LIN {X 0,Y 282.772,Z 519.685,A -85,B 0,C 180,E1 -19007.378,E2 -19007.378} C_VEL
LIN {X 0,Y 274.139,Z 501.017,A -85,B 0,C 180,E1 -19009.361,E2 -19009.361} C_VEL
LIN {X 0,Y 269.394,Z 492.351,A -85,B 0,C 180,E1 -19010.462,E2 -19010.462} C_VEL
LIN {X 0,Y 261.434,Z 479.486,A -85,B 0,C 180,E1 -19012.375,E2 -19012.375} C_VEL
LIN {X 0,Y 254.128,Z 468.54,A -85,B 0,C 180,E1 -19014.24,E2 -19014.24} C_VEL
LIN {X 0,Y 251.383,Z 464.398,A -85,B 0,C 180,E1 -19014.979,E2 -19014.979} C_VEL
LIN {X 0,Y 249.654,Z 462.021,A -85,B 0,C 180,E1 -19015.449,E2 -19015.449} C_VEL
LIN {X 0,Y 249.116,Z 460.076,A -85,B 0,C 180,E1 -19015.694,E2 -19015.694} C_VEL
LIN {X 0,Y 249.078,Z 460.074,A -85,B 0,C 180,E1 -19018.99,E2 -19018.99} C_VEL
LIN {X 0,Y 249.037,Z 460.072,A -85,B 0,C 180,E1 -19022.426,E2 -19022.426} C_VEL
LIN {X 0,Y 249.061,Z 460.079,A -85,B 0,C 180,E1 -19026.341,E2 -19026.341} C_VEL
LIN {X 0,Y 249.035,Z 460.089,A -85,B 0,C 180,E1 -19030.473,E2 -19030.473} C_VEL
LIN {X 0,Y 249.008,Z 460.09,A -85,B 0,C 180,E1 -19034.878,E2 -19034.878} C_VEL
LIN {X 0,Y 249.033,Z 460.078,A -85,B 0,C 180,E1 -19037.366,E2 -19037.366} C_VEL
LIN {X 0,Y 249.051,Z 460.087,A -85,B 0,C 180,E1 -19041.623,E2 -19041.623} C_VEL
LIN {X 0,Y 249.064,Z 460.077,A -85,B 0,C 180,E1 -19045.642,E2 -19045.642} C_VEL
LIN {X 0,Y 249.05,Z 460.069,A -85,B 0,C 180,E1 -19049.472,E2 -19049.472} C_VEL
LIN {X 0,Y 249.071,Z 460.084,A -85,B 0,C 180,E1 -19053.161,E2 -19053.161} C_VEL
LIN {X 0,Y 249.064,Z 460.062,A -85,B 0,C 180,E1 -19056.731,E2 -19056.731} C_VEL
LIN {X 0,Y 249.112,Z 460.078,A -85,B 0,C 180,E1 -19060.211,E2 -19060.211} C_VEL
LIN {X 0,Y 249.245,Z 460.04,A -85,B 0,C 180,E1 -19063.622,E2 -19063.622} C_VEL
LIN {X 0,Y 249.194,Z 460.062,A -85,B 0,C 180,E1 -19066.352,E2 -19066.352} C_VEL
LIN {X 0,Y 248.614,Z 460.143,A -85,B 0,C 180,E1 -19067.703,E2 -19067.703} C_VEL
LIN {X 0,Y 245.972,Z 460.48,A -85,B 0,C 180,E1 -19069.912,E2 -19069.912} C_VEL
LIN {X 0,Y 242.807,Z 460.868,A -85,B 0,C 180,E1 -19072.63,E2 -19072.63} C_VEL
LIN {X 0,Y 242.4,Z 460.912,A -85,B 0,C 180,E1 -19073.568,E2 -19073.568} C_VEL
LIN {X 0,Y 242.638,Z 460.869,A -85,B 0,C 180,E1 -19078.34,E2 -19078.34} C_VEL
LIN {X 0,Y 242.638,Z 460.881,A -85,B 0,C 180,E1 -19081.659,E2 -19081.659} C_VEL
LIN {X 0,Y 242.435,Z 460.897,A -85,B 0,C 180,E1 -19086.658,E2 -19086.658} C_VEL
LIN {X 0,Y 242.316,Z 460.916,A -85,B 0,C 180,E1 -19090.021,E2 -19090.021} C_VEL
LIN {X 0,Y 242.168,Z 460.944,A -85,B 0,C 180,E1 -19095.14,E2 -19095.14} C_VEL
LIN {X 0,Y 242.08,Z 460.932,A -85,B 0,C 180,E1 -19098.623,E2 -19098.623} C_VEL
LIN {X 0,Y 242.051,Z 460.957,A -85,B 0,C 180,E1 -19102.176,E2 -19102.176} C_VEL
LIN {X 0,Y 242.068,Z 460.953,A -85,B 0,C 180,E1 -19105.838,E2 -19105.838} C_VEL
LIN {X 0,Y 242.03,Z 460.962,A -85,B 0,C 180,E1 -19109.58,E2 -19109.58} C_VEL
LIN {X 0,Y 241.992,Z 460.962,A -85,B 0,C 180,E1 -19113.49,E2 -19113.49} C_VEL
LIN {X 0,Y 242.004,Z 460.963,A -85,B 0,C 180,E1 -19117.579,E2 -19117.579} C_VEL
LIN {X 0,Y 242.025,Z 461.128,A -85,B 0,C 180,E1 -19118.864,E2 -19118.864} C_VEL
LIN {X 0,Y 243.467,Z 465.75,A -85,B 0,C 180,E1 -19120.909,E2 -19120.909} C_VEL
LIN {X 0,Y 246.199,Z 470.197,A -85,B 0,C 180,E1 -19121.719,E2 -19121.719} C_VEL
LIN {X 0,Y 254.135,Z 483.567,A -85,B 0,C 180,E1 -19123.939,E2 -19123.939} C_VEL
LIN {X 0,Y 261.128,Z 496.498,A -85,B 0,C 180,E1 -19125.79,E2 -19125.79} C_VEL
LIN {X 0,Y 268.709,Z 512.001,A -85,B 0,C 180,E1 -19127.704,E2 -19127.704} C_VEL
LIN {X 0,Y 276.684,Z 530.632,A -85,B 0,C 180,E1 -19129.643,E2 -19129.643} C_VEL
LIN {X 0,Y 271.867,Z 629.009,A -85,B 0,C 180,E1 -19132.182,E2 -19132.182} C_VEL
LIN {X 0,Y 270.488,Z 644.739,A -85,B 0,C 180,E1 -19132.777,E2 -19132.777} C_VEL
LIN {X 0,Y 268.53,Z 659.205,A -85,B 0,C 180,E1 -19133.574,E2 -19133.574} C_VEL
LIN {X 0,Y 266.005,Z 673.975,A -85,B 0,C 180,E1 -19134.686,E2 -19134.686} C_VEL
LIN {X 0,Y 263.095,Z 688.32,A -85,B 0,C 180,E1 -19136.107,E2 -19136.107} C_VEL
LIN {X 0,Y 259.931,Z 701.339,A -85,B 0,C 180,E1 -19137.723,E2 -19137.723} C_VEL
LIN {X 0,Y 256.518,Z 714.469,A -85,B 0,C 180,E1 -19139.772,E2 -19139.772} C_VEL
LIN {X 0,Y 253.224,Z 725.427,A -85,B 0,C 180,E1 -19141.847,E2 -19141.847} C_VEL
LIN {X 0,Y 250.049,Z 736.273,A -85,B 0,C 180,E1 -19144.382,E2 -19144.382} C_VEL
LIN {X 0,Y 247.729,Z 744.182,A -85,B 0,C 180,E1 -19146.598,E2 -19146.598} C_VEL
LIN {X 0,Y 245.105,Z 752.602,A -85,B 0,C 180,E1 -19149.436,E2 -19149.436} C_VEL
LIN {X 0,Y 242.764,Z 760.654,A -85,B 0,C 180,E1 -19152.812,E2 -19152.812} C_VEL
LIN {X 0,Y 241.46,Z 766.039,A -85,B 0,C 180,E1 -19155.675,E2 -19155.675} C_VEL
LIN {X 0,Y 240.394,Z 771.037,A -85,B 0,C 180,E1 -19159.045,E2 -19159.045} C_VEL
LIN {X 0,Y 240.012,Z 773.943,A -85,B 0,C 180,E1 -19161.58,E2 -19161.58} C_VEL
LIN {X 0,Y 239.767,Z 776.64,A -85,B 0,C 180,E1 -19164.954,E2 -19164.954} C_VEL
LIN {X 0,Y 239.828,Z 778.136,A -85,B 0,C 180,E1 -19168.32,E2 -19168.32} C_VEL
LIN {X 0,Y 239.912,Z 778.446,A -85,B 0,C 180,E1 -19169.999,E2 -19169.999} C_VEL
LIN {X 0,Y 239.745,Z 778.19,A -85,B 0,C 180,E1 -19173.36,E2 -19173.36} C_VEL
LIN {X 0,Y 239.837,Z 776.785,A -85,B 0,C 180,E1 -19176.73,E2 -19176.73} C_VEL
LIN {X 0,Y 240.251,Z 774.162,A -85,B 0,C 180,E1 -19180.108,E2 -19180.108} C_VEL
LIN {X 0,Y 241.234,Z 770.329,A -85,B 0,C 180,E1 -19183.477,E2 -19183.477} C_VEL
LIN {X 0,Y 242.731,Z 765.203,A -85,B 0,C 180,E1 -19186.829,E2 -19186.829} C_VEL
LIN {X 0,Y 245.031,Z 758.665,A -85,B 0,C 180,E1 -19190.131,E2 -19190.131} C_VEL
LIN {X 0,Y 248.034,Z 750.541,A -85,B 0,C 180,E1 -19193.37,E2 -19193.37} C_VEL
LIN {X 0,Y 251.407,Z 741.915,A -85,B 0,C 180,E1 -19196.121,E2 -19196.121} C_VEL
LIN {X 0,Y 254.509,Z 733.203,A -85,B 0,C 180,E1 -19198.445,E2 -19198.445} C_VEL
LIN {X 0,Y 258.211,Z 722.949,A -85,B 0,C 180,E1 -19200.685,E2 -19200.685} C_VEL
LIN {X 0,Y 262.278,Z 710.731,A -85,B 0,C 180,E1 -19202.861,E2 -19202.861} C_VEL
LIN {X 0,Y 266.371,Z 697.186,A -85,B 0,C 180,E1 -19204.788,E2 -19204.788} C_VEL
LIN {X 0,Y 269.906,Z 683.486,A -85,B 0,C 180,E1 -19206.352,E2 -19206.352} C_VEL
LIN {X 0,Y 273.177,Z 668.696,A -85,B 0,C 180,E1 -19207.661,E2 -19207.661} C_VEL
LIN {X 0,Y 275.927,Z 654.171,A -85,B 0,C 180,E1 -19208.609,E2 -19208.609} C_VEL
LIN {X 0,Y 277.96,Z 639.385,A -85,B 0,C 180,E1 -19209.321,E2 -19209.321} C_VEL
LIN {X 0,Y 279.307,Z 622.797,A -85,B 0,C 180,E1 -19209.854,E2 -19209.854} C_VEL
LIN {X 0,Y 284.003,Z 540.814,A -85,B 0,C 180,E1 -19211.923,E2 -19211.923} C_VEL
LIN {X 0,Y 284.239,Z 534.234,A -85,B 0,C 180,E1 -19212.118,E2 -19212.118} C_VEL
LIN {X 0,Y 278.658,Z 520.932,A -85,B 0,C 180,E1 -19213.847,E2 -19213.847} C_VEL
LIN {X 0,Y 272.663,Z 508.788,A -85,B 0,C 180,E1 -19215.785,E2 -19215.785} C_VEL
LIN {X 0,Y 266.889,Z 498.341,A -85,B 0,C 180,E1 -19217.779,E2 -19217.779} C_VEL
LIN {X 0,Y 261.979,Z 490.421,A -85,B 0,C 180,E1 -19219.607,E2 -19219.607} C_VEL
LIN {X 0,Y 259.385,Z 486.385,A -85,B 0,C 180,E1 -19220.641,E2 -19220.641} C_VEL
LIN {X 0,Y 256.055,Z 481.339,A -85,B 0,C 180,E1 -19222.035,E2 -19222.035} C_VEL
LIN {X 0,Y 251.669,Z 475.022,A -85,B 0,C 180,E1 -19224.04,E2 -19224.04} C_VEL
LIN {X 0,Y 248.15,Z 470.216,A -85,B 0,C 180,E1 -19225.806,E2 -19225.806} C_VEL
LIN {X 0,Y 244.223,Z 465.374,A -85,B 0,C 180,E1 -19227.948,E2 -19227.948} C_VEL
LIN {X 0,Y 242.555,Z 462.973,A -85,B 0,C 180,E1 -19229.05,E2 -19229.05} C_VEL
LIN {X 0,Y 242.027,Z 460.958,A -85,B 0,C 180,E1 -19230.752,E2 -19230.752} C_VEL
LIN {X 0,Y 242.062,Z 460.956,A -85,B 0,C 180,E1 -19234.183,E2 -19234.183} C_VEL
LIN {X 0,Y 242.047,Z 460.958,A -85,B 0,C 180,E1 -19238.297,E2 -19238.297} C_VEL
LIN {X 0,Y 242.157,Z 460.935,A -85,B 0,C 180,E1 -19243.278,E2 -19243.278} C_VEL
LIN {X 0,Y 242.181,Z 460.942,A -85,B 0,C 180,E1 -19248.28,E2 -19248.28} C_VEL
LIN {X 0,Y 242.422,Z 460.909,A -85,B 0,C 180,E1 -19251.666,E2 -19251.666} C_VEL
LIN {X 0,Y 242.256,Z 460.926,A -85,B 0,C 180,E1 -19255.008,E2 -19255.008} C_VEL
LIN {X 0,Y 242.631,Z 460.878,A -85,B 0,C 180,E1 -19258.341,E2 -19258.341} C_VEL
LIN {X 0,Y 242.631,Z 460.877,A -85,B 0,C 180,E1 -19261.66,E2 -19261.66} C_VEL
LIN {X 0,Y 242.425,Z 460.912,A -85,B 0,C 180,E1 -19266.706,E2 -19266.706} C_VEL
LIN {X 0,Y 242.406,Z 461.074,A -85,B 0,C 180,E1 -19269.237,E2 -19269.237} C_VEL
LIN {X 0,Y 243.246,Z 463.656,A -85,B 0,C 180,E1 -19269.881,E2 -19269.881} C_VEL
LIN {X 0,Y 245.242,Z 465.908,A -85,B 0,C 180,E1 -19271.049,E2 -19271.049} C_VEL
LIN {X 0,Y 246.841,Z 466.95,A -85,B 0,C 180,E1 -19271.861,E2 -19271.861} C_VEL
LIN {X 0,Y 248.548,Z 470.005,A -85,B 0,C 180,E1 -19272.815,E2 -19272.815} C_VEL
LIN {X 0,Y 251.376,Z 472.668,A -85,B 0,C 180,E1 -19274.161,E2 -19274.161} C_VEL
LIN {X 0,Y 253.704,Z 476.012,A -85,B 0,C 180,E1 -19275.273,E2 -19275.273} C_VEL
LIN {X 0,Y 255.328,Z 477.907,A -85,B 0,C 180,E1 -19275.978,E2 -19275.978} C_VEL
LIN {X 0,Y 258.103,Z 481.555,A -85,B 0,C 180,E1 -19277.142,E2 -19277.142} C_VEL
LIN {X 0,Y 262.643,Z 487.86,A -85,B 0,C 180,E1 -19278.933,E2 -19278.933} C_VEL
LIN {X 0,Y 267.991,Z 495.314,A -85,B 0,C 180,E1 -19280.849,E2 -19280.849} C_VEL
LIN {X 0,Y 273.848,Z 504.485,A -85,B 0,C 180,E1 -19282.791,E2 -19282.791} C_VEL
LIN {X 0,Y 280.321,Z 516.959,A -85,B 0,C 180,E1 -19284.831,E2 -19284.831} C_VEL
LIN {X 0,Y 284.68,Z 526.585,A -85,B 0,C 180,E1 -19286.148,E2 -19286.148} C_VEL
LIN {X 0,Y 279.259,Z 620.067,A -85,B 0,C 180,E1 -19288.545,E2 -19288.545} C_VEL
LIN {X 0,Y 277.451,Z 636.178,A -85,B 0,C 180,E1 -19289.197,E2 -19289.197} C_VEL
LIN {X 0,Y 275.126,Z 651.64,A -85,B 0,C 180,E1 -19290.15,E2 -19290.15} C_VEL
LIN {X 0,Y 272.338,Z 665.875,A -85,B 0,C 180,E1 -19291.316,E2 -19291.316} C_VEL
LIN {X 0,Y 268.818,Z 680.57,A -85,B 0,C 180,E1 -19292.875,E2 -19292.875} C_VEL
LIN {X 0,Y 264.966,Z 694.127,A -85,B 0,C 180,E1 -19294.692,E2 -19294.692} C_VEL
LIN {X 0,Y 261.065,Z 706.563,A -85,B 0,C 180,E1 -19296.788,E2 -19296.788} C_VEL
LIN {X 0,Y 257.532,Z 716.783,A -85,B 0,C 180,E1 -19298.879,E2 -19298.879} C_VEL
LIN {X 0,Y 253.615,Z 727.436,A -85,B 0,C 180,E1 -19301.567,E2 -19301.567} C_VEL
LIN {X 0,Y 250.381,Z 735.735,A -85,B 0,C 180,E1 -19304.125,E2 -19304.125} C_VEL
LIN {X 0,Y 247.359,Z 743.322,A -85,B 0,C 180,E1 -19307.01,E2 -19307.01} C_VEL
LIN {X 0,Y 244.99,Z 749.256,A -85,B 0,C 180,E1 -19309.802,E2 -19309.802} C_VEL
LIN {X 0,Y 243.157,Z 754.125,A -85,B 0,C 180,E1 -19312.631,E2 -19312.631} C_VEL
LIN {X 0,Y 241.771,Z 757.966,A -85,B 0,C 180,E1 -19315.471,E2 -19315.471} C_VEL
LIN {X 0,Y 240.791,Z 760.856,A -85,B 0,C 180,E1 -19318.309,E2 -19318.309} C_VEL
LIN {X 0,Y 239.89,Z 763.38,A -85,B 0,C 180,E1 -19322.048,E2 -19322.048} C_VEL
LIN {X 0,Y 239.488,Z 764.479,A -85,B 0,C 180,E1 -19325.744,E2 -19325.744} C_VEL
LIN {X 0,Y 239.448,Z 764.232,A -85,B 0,C 180,E1 -19329.379,E2 -19329.379} C_VEL
LIN {X 0,Y 239.694,Z 762.699,A -85,B 0,C 180,E1 -19332.951,E2 -19332.951} C_VEL
LIN {X 0,Y 240.343,Z 759.891,A -85,B 0,C 180,E1 -19336.472,E2 -19336.472} C_VEL
LIN {X 0,Y 241.291,Z 755.788,A -85,B 0,C 180,E1 -19339.936,E2 -19339.936} C_VEL
LIN {X 0,Y 242.794,Z 750.301,A -85,B 0,C 180,E1 -19343.352,E2 -19343.352} C_VEL
LIN {X 0,Y 244.872,Z 743.309,A -85,B 0,C 180,E1 -19346.71,E2 -19346.71} C_VEL
LIN {X 0,Y 247.209,Z 735.768,A -85,B 0,C 180,E1 -19349.594,E2 -19349.594} C_VEL
LIN {X 0,Y 250.045,Z 726.708,A -85,B 0,C 180,E1 -19352.417,E2 -19352.417} C_VEL
LIN {X 0,Y 252.897,Z 717.459,A -85,B 0,C 180,E1 -19354.783,E2 -19354.783} C_VEL
LIN {X 0,Y 256.069,Z 706.558,A -85,B 0,C 180,E1 -19357.095,E2 -19357.095} C_VEL
LIN {X 0,Y 259.336,Z 694.632,A -85,B 0,C 180,E1 -19359.162,E2 -19359.162} C_VEL
LIN {X 0,Y 262.573,Z 681.588,A -85,B 0,C 180,E1 -19360.995,E2 -19360.995} C_VEL
LIN {X 0,Y 265.303,Z 668.808,A -85,B 0,C 180,E1 -19362.449,E2 -19362.449} C_VEL
LIN {X 0,Y 267.697,Z 655.458,A -85,B 0,C 180,E1 -19363.668,E2 -19363.668} C_VEL
LIN {X 0,Y 269.882,Z 640.363,A -85,B 0,C 180,E1 -19364.718,E2 -19364.718} C_VEL
LIN {X 0,Y 271.473,Z 626.008,A -85,B 0,C 180,E1 -19365.437,E2 -19365.437} C_VEL
LIN {X 0,Y 272.537,Z 610.439,A -85,B 0,C 180,E1 -19365.951,E2 -19365.951} C_VEL
LIN {X 0,Y 276.972,Z 521.758,A -85,B 0,C 180,E1 -19368.204,E2 -19368.204} C_VEL
LIN {X 0,Y 268.071,Z 502.626,A -85,B 0,C 180,E1 -19370.328,E2 -19370.328} C_VEL
LIN {X 0,Y 260.016,Z 488.824,A -85,B 0,C 180,E1 -19372.298,E2 -19372.298} C_VEL
LIN {X 0,Y 250.255,Z 473.861,A -85,B 0,C 180,E1 -19374.84,E2 -19374.84} C_VEL
LIN {X 0,Y 246.987,Z 469.165,A -85,B 0,C 180,E1 -19375.744,E2 -19375.744} C_VEL
LIN {X 0,Y 244.718,Z 465.681,A -85,B 0,C 180,E1 -19376.405,E2 -19376.405} C_VEL
LIN {X 0,Y 242.781,Z 463.346,A -85,B 0,C 180,E1 -19376.953,E2 -19376.953} C_VEL
LIN {X 0,Y 242.02,Z 460.953,A -85,B 0,C 180,E1 -19377.294,E2 -19377.294} C_VEL
LIN {X 0,Y 241.977,Z 460.958,A -85,B 0,C 180,E1 -19381.52,E2 -19381.52} C_VEL
LIN {X 0,Y 242.009,Z 460.965,A -85,B 0,C 180,E1 -19385.597,E2 -19385.597} C_VEL
LIN {X 0,Y 241.979,Z 460.959,A -85,B 0,C 180,E1 -19389.715,E2 -19389.715} C_VEL
LIN {X 0,Y 241.937,Z 460.963,A -85,B 0,C 180,E1 -19394.201,E2 -19394.201} C_VEL
LIN {X 0,Y 241.957,Z 460.954,A -85,B 0,C 180,E1 -19398.081,E2 -19398.081} C_VEL
LIN {X 0,Y 242.014,Z 460.958,A -85,B 0,C 180,E1 -19402.422,E2 -19402.422} C_VEL
LIN {X 0,Y 241.994,Z 460.966,A -85,B 0,C 180,E1 -19406.509,E2 -19406.509} C_VEL
LIN {X 0,Y 242.016,Z 460.944,A -85,B 0,C 180,E1 -19410.597,E2 -19410.597} C_VEL
LIN {X 0,Y 242.071,Z 460.954,A -85,B 0,C 180,E1 -19414.183,E2 -19414.183} C_VEL
LIN {X 0,Y 242.029,Z 460.95,A -85,B 0,C 180,E1 -19418.313,E2 -19418.313} C_VEL
LIN {X 0,Y 242.166,Z 460.921,A -85,B 0,C 180,E1 -19423.278,E2 -19423.278} C_VEL
LIN {X 0,Y 242.189,Z 460.934,A -85,B 0,C 180,E1 -19428.279,E2 -19428.279} C_VEL
LIN {X 0,Y 242.43,Z 460.896,A -85,B 0,C 180,E1 -19431.665,E2 -19431.665} C_VEL
LIN {X 0,Y 242.4,Z 460.912,A -85,B 0,C 180,E1 -19433.568,E2 -19433.568} C_VEL
LIN {X 0,Y 241.633,Z 461.006,A -85,B 0,C 180,E1 -19434.956,E2 -19434.956} C_VEL
LIN {X 0,Y 238.895,Z 461.343,A -85,B 0,C 180,E1 -19437.229,E2 -19437.229} C_VEL
LIN {X 0,Y 235.898,Z 461.726,A -85,B 0,C 180,E1 -19440.028,E2 -19440.028} C_VEL
LIN {X 0,Y 235.597,Z 461.756,A -85,B 0,C 180,E1 -19440.993,E2 -19440.993} C_VEL
LIN {X 0,Y 235.406,Z 461.776,A -85,B 0,C 180,E1 -19446.858,E2 -19446.858} C_VEL
LIN {X 0,Y 235.24,Z 461.792,A -85,B 0,C 180,E1 -19450.326,E2 -19450.326} C_VEL
LIN {X 0,Y 235.115,Z 461.824,A -85,B 0,C 180,E1 -19455.606,E2 -19455.606} C_VEL
LIN {X 0,Y 235.021,Z 461.812,A -85,B 0,C 180,E1 -19459.204,E2 -19459.204} C_VEL
LIN {X 0,Y 234.982,Z 461.835,A -85,B 0,C 180,E1 -19462.88,E2 -19462.88} C_VEL
LIN {X 0,Y 234.971,Z 461.841,A -85,B 0,C 180,E1 -19466.657,E2 -19466.657} C_VEL
LIN {X 0,Y 234.933,Z 461.842,A -85,B 0,C 180,E1 -19470.567,E2 -19470.567} C_VEL
LIN {X 0,Y 234.962,Z 461.843,A -85,B 0,C 180,E1 -19474.632,E2 -19474.632} C_VEL
LIN {X 0,Y 234.993,Z 461.954,A -85,B 0,C 180,E1 -19477.475,E2 -19477.475} C_VEL
LIN {X 0,Y 236.086,Z 465.459,A -85,B 0,C 180,E1 -19479.1,E2 -19479.1} C_VEL
LIN {X 0,Y 238.996,Z 470.175,A -85,B 0,C 180,E1 -19480.035,E2 -19480.035} C_VEL
LIN {X 0,Y 244.121,Z 478.587,A -85,B 0,C 180,E1 -19481.601,E2 -19481.601} C_VEL
LIN {X 0,Y 251.332,Z 490.98,A -85,B 0,C 180,E1 -19483.658,E2 -19483.658} C_VEL
LIN {X 0,Y 257.649,Z 503.054,A -85,B 0,C 180,E1 -19485.379,E2 -19485.379} C_VEL
LIN {X 0,Y 264.473,Z 517.44,A -85,B 0,C 180,E1 -19487.163,E2 -19487.163} C_VEL
LIN {X 0,Y 270.998,Z 532.796,A -85,B 0,C 180,E1 -19488.807,E2 -19488.807} C_VEL
LIN {X 0,Y 265.95,Z 630.58,A -85,B 0,C 180,E1 -19491.368,E2 -19491.368} C_VEL
LIN {X 0,Y 264.511,Z 645.629,A -85,B 0,C 180,E1 -19491.968,E2 -19491.968} C_VEL
LIN {X 0,Y 262.408,Z 660.442,A -85,B 0,C 180,E1 -19492.822,E2 -19492.822} C_VEL
LIN {X 0,Y 259.934,Z 674.242,A -85,B 0,C 180,E1 -19493.896,E2 -19493.896} C_VEL
LIN {X 0,Y 257.031,Z 687.913,A -85,B 0,C 180,E1 -19495.269,E2 -19495.269} C_VEL
LIN {X 0,Y 253.55,Z 701.866,A -85,B 0,C 180,E1 -19497.045,E2 -19497.045} C_VEL
LIN {X 0,Y 250.338,Z 713.789,A -85,B 0,C 180,E1 -19498.944,E2 -19498.944} C_VEL
LIN {X 0,Y 246.913,Z 724.827,A -85,B 0,C 180,E1 -19501.06,E2 -19501.06} C_VEL
LIN {X 0,Y 243.716,Z 735.267,A -85,B 0,C 180,E1 -19503.522,E2 -19503.522} C_VEL
LIN {X 0,Y 241.164,Z 743.679,A -85,B 0,C 180,E1 -19505.921,E2 -19505.921} C_VEL
LIN {X 0,Y 238.39,Z 752.151,A -85,B 0,C 180,E1 -19508.829,E2 -19508.829} C_VEL
LIN {X 0,Y 236.203,Z 759.359,A -85,B 0,C 180,E1 -19511.884,E2 -19511.884} C_VEL
LIN {X 0,Y 234.506,Z 765.677,A -85,B 0,C 180,E1 -19515.241,E2 -19515.241} C_VEL
LIN {X 0,Y 233.376,Z 770.716,A -85,B 0,C 180,E1 -19518.711,E2 -19518.711} C_VEL
LIN {X 0,Y 232.94,Z 773.639,A -85,B 0,C 180,E1 -19521.323,E2 -19521.323} C_VEL
LIN {X 0,Y 232.686,Z 776.373,A -85,B 0,C 180,E1 -19524.8,E2 -19524.8} C_VEL
LIN {X 0,Y 232.739,Z 777.903,A -85,B 0,C 180,E1 -19528.269,E2 -19528.269} C_VEL
LIN {X 0,Y 232.822,Z 778.23,A -85,B 0,C 180,E1 -19529.999,E2 -19529.999} C_VEL
LIN {X 0,Y 232.653,Z 778.005,A -85,B 0,C 180,E1 -19533.463,E2 -19533.463} C_VEL
LIN {X 0,Y 232.765,Z 776.622,A -85,B 0,C 180,E1 -19536.936,E2 -19536.936} C_VEL
LIN {X 0,Y 233.198,Z 774.024,A -85,B 0,C 180,E1 -19540.417,E2 -19540.417} C_VEL
LIN {X 0,Y 234.262,Z 770.229,A -85,B 0,C 180,E1 -19543.886,E2 -19543.886} C_VEL
LIN {X 0,Y 235.864,Z 765.15,A -85,B 0,C 180,E1 -19547.334,E2 -19547.334} C_VEL
LIN {X 0,Y 238.306,Z 758.66,A -85,B 0,C 180,E1 -19550.725,E2 -19550.725} C_VEL
LIN {X 0,Y 241.497,Z 750.583,A -85,B 0,C 180,E1 -19554.042,E2 -19554.042} C_VEL
LIN {X 0,Y 244.976,Z 742.009,A -85,B 0,C 180,E1 -19556.861,E2 -19556.861} C_VEL
LIN {X 0,Y 248.88,Z 731.737,A -85,B 0,C 180,E1 -19559.614,E2 -19559.614} C_VEL
LIN {X 0,Y 252.791,Z 721.28,A -85,B 0,C 180,E1 -19561.885,E2 -19561.885} C_VEL
LIN {X 0,Y 256.718,Z 709.956,A -85,B 0,C 180,E1 -19563.902,E2 -19563.902} C_VEL
LIN {X 0,Y 260.597,Z 697.687,A -85,B 0,C 180,E1 -19565.675,E2 -19565.675} C_VEL
LIN {X 0,Y 264.24,Z 684.24,A -85,B 0,C 180,E1 -19567.247,E2 -19567.247} C_VEL
LIN {X 0,Y 267.634,Z 669.612,A -85,B 0,C 180,E1 -19568.583,E2 -19568.583} C_VEL
LIN {X 0,Y 270.451,Z 655.394,A -85,B 0,C 180,E1 -19569.542,E2 -19569.542} C_VEL
LIN {X 0,Y 272.679,Z 640.192,A -85,B 0,C 180,E1 -19570.296,E2 -19570.296} C_VEL
LIN {X 0,Y 274.085,Z 624.371,A -85,B 0,C 180,E1 -19570.832,E2 -19570.832} C_VEL
LIN {X 0,Y 278.869,Z 544.481,A -85,B 0,C 180,E1 -19572.877,E2 -19572.877} C_VEL
LIN {X 0,Y 279.189,Z 536.605,A -85,B 0,C 180,E1 -19573.113,E2 -19573.113} C_VEL
LIN {X 0,Y 274.25,Z 524.669,A -85,B 0,C 180,E1 -19574.724,E2 -19574.724} C_VEL
LIN {X 0,Y 267.81,Z 511.374,A -85,B 0,C 180,E1 -19576.94,E2 -19576.94} C_VEL
LIN {X 0,Y 262.063,Z 501.21,A -85,B 0,C 180,E1 -19579.053,E2 -19579.053} C_VEL
LIN {X 0,Y 257.009,Z 492.813,A -85,B 0,C 180,E1 -19581.095,E2 -19581.095} C_VEL
LIN {X 0,Y 252.965,Z 486.736,A -85,B 0,C 180,E1 -19582.854,E2 -19582.854} C_VEL
LIN {X 0,Y 249.079,Z 480.95,A -85,B 0,C 180,E1 -19584.732,E2 -19584.732} C_VEL
LIN {X 0,Y 244.987,Z 475.331,A -85,B 0,C 180,E1 -19586.888,E2 -19586.888} C_VEL
LIN {X 0,Y 239.896,Z 468.74,A -85,B 0,C 180,E1 -19590.009,E2 -19590.009} C_VEL
LIN {X 0,Y 238.059,Z 466.791,A -85,B 0,C 180,E1 -19591.253,E2 -19591.253} C_VEL
LIN {X 0,Y 236.004,Z 464.746,A -85,B 0,C 180,E1 -19592.752,E2 -19592.752} C_VEL
LIN {X 0,Y 235.076,Z 462.308,A -85,B 0,C 180,E1 -19593.75,E2 -19593.75} C_VEL
LIN {X 0,Y 235.017,Z 461.836,A -85,B 0,C 180,E1 -19594.499,E2 -19594.499} C_VEL
LIN {X 0,Y 235.005,Z 461.829,A -85,B 0,C 180,E1 -19598.97,E2 -19598.97} C_VEL
LIN {X 0,Y 235.091,Z 461.815,A -85,B 0,C 180,E1 -19603.059,E2 -19603.059} C_VEL
LIN {X 0,Y 235.113,Z 461.818,A -85,B 0,C 180,E1 -19607.922,E2 -19607.922} C_VEL
LIN {X 0,Y 235.371,Z 461.784,A -85,B 0,C 180,E1 -19611.414,E2 -19611.414} C_VEL
LIN {X 0,Y 235.399,Z 461.781,A -85,B 0,C 180,E1 -19613.142,E2 -19613.142} C_VEL
LIN {X 0,Y 235.591,Z 461.754,A -85,B 0,C 180,E1 -19618.291,E2 -19618.291} C_VEL
LIN {X 0,Y 235.591,Z 461.754,A -85,B 0,C 180,E1 -19621.71,E2 -19621.71} C_VEL
LIN {X 0,Y 235.231,Z 461.943,A -85,B 0,C 180,E1 -19624.874,E2 -19624.874} C_VEL
LIN {X 0,Y 235.951,Z 464.084,A -85,B 0,C 180,E1 -19625.609,E2 -19625.609} C_VEL
LIN {X 0,Y 238.09,Z 466.548,A -85,B 0,C 180,E1 -19627.207,E2 -19627.207} C_VEL
LIN {X 0,Y 240.259,Z 467.791,A -85,B 0,C 180,E1 -19628.581,E2 -19628.581} C_VEL
LIN {X 0,Y 241.66,Z 470.698,A -85,B 0,C 180,E1 -19629.578,E2 -19629.578} C_VEL
LIN {X 0,Y 244.287,Z 473.107,A -85,B 0,C 180,E1 -19631.093,E2 -19631.093} C_VEL
LIN {X 0,Y 247.164,Z 477.235,A -85,B 0,C 180,E1 -19632.679,E2 -19632.679} C_VEL
LIN {X 0,Y 249.087,Z 479.099,A -85,B 0,C 180,E1 -19633.617,E2 -19633.617} C_VEL
LIN {X 0,Y 251.81,Z 482.758,A -85,B 0,C 180,E1 -19634.937,E2 -19634.937} C_VEL
LIN {X 0,Y 256.792,Z 489.477,A -85,B 0,C 180,E1 -19637.117,E2 -19637.117} C_VEL
LIN {X 0,Y 262.812,Z 498.023,A -85,B 0,C 180,E1 -19639.478,E2 -19639.478} C_VEL
LIN {X 0,Y 268.738,Z 507.04,A -85,B 0,C 180,E1 -19641.577,E2 -19641.577} C_VEL
LIN {X 0,Y 274.345,Z 517.578,A -85,B 0,C 180,E1 -19643.465,E2 -19643.465} C_VEL
LIN {X 0,Y 279.611,Z 528.887,A -85,B 0,C 180,E1 -19645.139,E2 -19645.139} C_VEL
LIN {X 0,Y 274.128,Z 620.295,A -85,B 0,C 180,E1 -19647.529,E2 -19647.529} C_VEL
LIN {X 0,Y 272.323,Z 636.028,A -85,B 0,C 180,E1 -19648.172,E2 -19648.172} C_VEL
LIN {X 0,Y 269.96,Z 651.279,A -85,B 0,C 180,E1 -19649.107,E2 -19649.107} C_VEL
LIN {X 0,Y 266.818,Z 666.703,A -85,B 0,C 180,E1 -19650.389,E2 -19650.389} C_VEL
LIN {X 0,Y 263.465,Z 680.303,A -85,B 0,C 180,E1 -19651.848,E2 -19651.848} C_VEL
LIN {X 0,Y 259.55,Z 693.614,A -85,B 0,C 180,E1 -19653.632,E2 -19653.632} C_VEL
LIN {X 0,Y 255.93,Z 704.914,A -85,B 0,C 180,E1 -19655.52,E2 -19655.52} C_VEL
LIN {X 0,Y 251.674,Z 716.605,A -85,B 0,C 180,E1 -19657.905,E2 -19657.905} C_VEL
LIN {X 0,Y 247.672,Z 727.043,A -85,B 0,C 180,E1 -19660.565,E2 -19660.565} C_VEL
LIN {X 0,Y 244.033,Z 735.932,A -85,B 0,C 180,E1 -19663.351,E2 -19663.351} C_VEL
LIN {X 0,Y 240.717,Z 743.827,A -85,B 0,C 180,E1 -19666.429,E2 -19666.429} C_VEL
LIN {X 0,Y 238.071,Z 750.096,A -85,B 0,C 180,E1 -19669.501,E2 -19669.501} C_VEL
LIN {X 0,Y 236.156,Z 754.814,A -85,B 0,C 180,E1 -19672.407,E2 -19672.407} C_VEL
LIN {X 0,Y 234.733,Z 758.576,A -85,B 0,C 180,E1 -19675.33,E2 -19675.33} C_VEL
LIN {X 0,Y 234.029,Z 760.54,A -85,B 0,C 180,E1 -19677.281,E2 -19677.281} C_VEL
LIN {X 0,Y 232.954,Z 763.307,A -85,B 0,C 180,E1 -19681.139,E2 -19681.139} C_VEL
LIN {X 0,Y 232.419,Z 764.636,A -85,B 0,C 180,E1 -19684.956,E2 -19684.956} C_VEL
LIN {X 0,Y 232.308,Z 764.599,A -85,B 0,C 180,E1 -19688.715,E2 -19688.715} C_VEL
LIN {X 0,Y 232.551,Z 763.252,A -85,B 0,C 180,E1 -19692.411,E2 -19692.411} C_VEL
LIN {X 0,Y 233.141,Z 760.632,A -85,B 0,C 180,E1 -19696.046,E2 -19696.046} C_VEL
LIN {X 0,Y 234.098,Z 756.726,A -85,B 0,C 180,E1 -19699.624,E2 -19699.624} C_VEL
LIN {X 0,Y 235.567,Z 751.469,A -85,B 0,C 180,E1 -19703.147,E2 -19703.147} C_VEL
LIN {X 0,Y 237.606,Z 744.741,A -85,B 0,C 180,E1 -19706.61,E2 -19706.61} C_VEL
LIN {X 0,Y 240.008,Z 737.369,A -85,B 0,C 180,E1 -19709.616,E2 -19709.616} C_VEL
LIN {X 0,Y 242.827,Z 728.716,A -85,B 0,C 180,E1 -19712.489,E2 -19712.489} C_VEL
LIN {X 0,Y 246.303,Z 718.004,A -85,B 0,C 180,E1 -19715.363,E2 -19715.363} C_VEL
LIN {X 0,Y 249.518,Z 707.369,A -85,B 0,C 180,E1 -19717.689,E2 -19717.689} C_VEL
LIN {X 0,Y 252.912,Z 695.548,A -85,B 0,C 180,E1 -19719.8,E2 -19719.8} C_VEL
LIN {X 0,Y 256.216,Z 682.661,A -85,B 0,C 180,E1 -19721.672,E2 -19721.672} C_VEL
LIN {X 0,Y 259.359,Z 668.478,A -85,B 0,C 180,E1 -19723.317,E2 -19723.317} C_VEL
LIN {X 0,Y 262.016,Z 653.89,A -85,B 0,C 180,E1 -19724.64,E2 -19724.64} C_VEL
LIN {X 0,Y 264.201,Z 638.736,A -85,B 0,C 180,E1 -19725.675,E2 -19725.675} C_VEL
LIN {X 0,Y 265.885,Z 623.254,A -85,B 0,C 180,E1 -19726.41,E2 -19726.41} C_VEL
LIN {X 0,Y 267.195,Z 602.123,A -85,B 0,C 180,E1 -19727.033,E2 -19727.033} C_VEL
LIN {X 0,Y 271.179,Z 523.87,A -85,B 0,C 180,E1 -19729.064,E2 -19729.064} C_VEL
LIN {X 0,Y 263.096,Z 506.355,A -85,B 0,C 180,E1 -19731.078,E2 -19731.078} C_VEL
LIN {X 0,Y 254.851,Z 492.324,A -85,B 0,C 180,E1 -19733.166,E2 -19733.166} C_VEL
LIN {X 0,Y 245.729,Z 478.276,A -85,B 0,C 180,E1 -19735.648,E2 -19735.648} C_VEL
LIN {X 0,Y 240.582,Z 470.787,A -85,B 0,C 180,E1 -19737.15,E2 -19737.15} C_VEL
LIN {X 0,Y 238.387,Z 467.61,A -85,B 0,C 180,E1 -19737.816,E2 -19737.816} C_VEL
LIN {X 0,Y 237.56,Z 466.5,A -85,B 0,C 180,E1 -19738.068,E2 -19738.068} C_VEL
LIN {X 0,Y 235.607,Z 464.055,A -85,B 0,C 180,E1 -19738.666,E2 -19738.666} C_VEL
LIN {X 0,Y 234.951,Z 461.833,A -85,B 0,C 180,E1 -19739.016,E2 -19739.016} C_VEL
LIN {X 0,Y 234.951,Z 461.827,A -85,B 0,C 180,E1 -19743.116,E2 -19743.116} C_VEL
LIN {X 0,Y 234.933,Z 461.831,A -85,B 0,C 180,E1 -19746.749,E2 -19746.749} C_VEL
LIN {X 0,Y 234.945,Z 461.826,A -85,B 0,C 180,E1 -19748.944,E2 -19748.944} C_VEL
LIN {X 0,Y 234.893,Z 461.837,A -85,B 0,C 180,E1 -19753.485,E2 -19753.485} C_VEL
LIN {X 0,Y 234.924,Z 461.845,A -85,B 0,C 180,E1 -19756.522,E2 -19756.522} C_VEL
LIN {X 0,Y 234.958,Z 461.843,A -85,B 0,C 180,E1 -19761.086,E2 -19761.086} C_VEL
LIN {X 0,Y 234.964,Z 461.831,A -85,B 0,C 180,E1 -19765.367,E2 -19765.367} C_VEL
LIN {X 0,Y 234.926,Z 461.828,A -85,B 0,C 180,E1 -19769.431,E2 -19769.431} C_VEL
LIN {X 0,Y 234.996,Z 461.837,A -85,B 0,C 180,E1 -19773.794,E2 -19773.794} C_VEL
LIN {X 0,Y 235.001,Z 461.833,A -85,B 0,C 180,E1 -19778.968,E2 -19778.968} C_VEL
LIN {X 0,Y 235.099,Z 461.802,A -85,B 0,C 180,E1 -19783.059,E2 -19783.059} C_VEL
LIN {X 0,Y 235.149,Z 461.813,A -85,B 0,C 180,E1 -19787.923,E2 -19787.923} C_VEL
LIN {X 0,Y 235.379,Z 461.771,A -85,B 0,C 180,E1 -19791.414,E2 -19791.414} C_VEL
LIN {X 0,Y 235.349,Z 461.789,A -85,B 0,C 180,E1 -19793.51,E2 -19793.51} C_VEL
LIN {X 0,Y 235.597,Z 461.745,A -85,B 0,C 180,E1 -19798.29,E2 -19798.29} C_VEL
LIN {X 0,Y 235.597,Z 461.756,A -85,B 0,C 180,E1 -19800.993,E2 -19800.993} C_VEL
LIN {X 0,Y 234.884,Z 461.842,A -85,B 0,C 180,E1 -19802.416,E2 -19802.416} C_VEL
LIN {X 0,Y 231.923,Z 462.206,A -85,B 0,C 180,E1 -19804.733,E2 -19804.733} C_VEL
LIN {X 0,Y 229.429,Z 462.517,A -85,B 0,C 180,E1 -19806.623,E2 -19806.623} C_VEL
LIN {X 0,Y 228.378,Z 462.663,A -85,B 0,C 180,E1 -19808.093,E2 -19808.093} C_VEL
LIN {X 0,Y 228.302,Z 462.668,A -85,B 0,C 180,E1 -19808.592,E2 -19808.592} C_VEL
LIN {X 0,Y 228.077,Z 462.672,A -85,B 0,C 180,E1 -19812.456,E2 -19812.456} C_VEL
LIN {X 0,Y 228.037,Z 462.689,A -85,B 0,C 180,E1 -19817.174,E2 -19817.174} C_VEL
LIN {X 0,Y 227.961,Z 462.712,A -85,B 0,C 180,E1 -19822.347,E2 -19822.347} C_VEL
LIN {X 0,Y 227.944,Z 462.715,A -85,B 0,C 180,E1 -19826.602,E2 -19826.602} C_VEL
LIN {X 0,Y 227.909,Z 462.718,A -85,B 0,C 180,E1 -19830.295,E2 -19830.295} C_VEL
LIN {X 0,Y 227.891,Z 462.719,A -85,B 0,C 180,E1 -19833.718,E2 -19833.718} C_VEL
LIN {X 0,Y 227.951,Z 462.886,A -85,B 0,C 180,E1 -19836.028,E2 -19836.028} C_VEL
LIN {X 0,Y 228.707,Z 465.217,A -85,B 0,C 180,E1 -19837.156,E2 -19837.156} C_VEL
LIN {X 0,Y 231.477,Z 469.647,A -85,B 0,C 180,E1 -19838.11,E2 -19838.11} C_VEL
LIN {X 0,Y 236.582,Z 477.781,A -85,B 0,C 180,E1 -19839.78,E2 -19839.78} C_VEL
LIN {X 0,Y 241.919,Z 486.668,A -85,B 0,C 180,E1 -19841.44,E2 -19841.44} C_VEL
LIN {X 0,Y 249.18,Z 499.721,A -85,B 0,C 180,E1 -19843.56,E2 -19843.56} C_VEL
LIN {X 0,Y 257.658,Z 516.902,A -85,B 0,C 180,E1 -19845.901,E2 -19845.901} C_VEL
LIN {X 0,Y 265.288,Z 534.93,A -85,B 0,C 180,E1 -19847.929,E2 -19847.929} C_VEL
LIN {X 0,Y 260.182,Z 630.385,A -85,B 0,C 180,E1 -19850.471,E2 -19850.471} C_VEL
LIN {X 0,Y 258.699,Z 645.428,A -85,B 0,C 180,E1 -19851.08,E2 -19851.08} C_VEL
LIN {X 0,Y 256.517,Z 660.233,A -85,B 0,C 180,E1 -19851.942,E2 -19851.942} C_VEL
LIN {X 0,Y 253.845,Z 674.742,A -85,B 0,C 180,E1 -19853.098,E2 -19853.098} C_VEL
LIN {X 0,Y 250.731,Z 688.757,A -85,B 0,C 180,E1 -19854.551,E2 -19854.551} C_VEL
LIN {X 0,Y 247.589,Z 701.022,A -85,B 0,C 180,E1 -19856.146,E2 -19856.146} C_VEL
LIN {X 0,Y 244.177,Z 713.055,A -85,B 0,C 180,E1 -19858.07,E2 -19858.07} C_VEL
LIN {X 0,Y 240.656,Z 724.191,A -85,B 0,C 180,E1 -19860.233,E2 -19860.233} C_VEL
LIN {X 0,Y 237.376,Z 734.36,A -85,B 0,C 180,E1 -19862.648,E2 -19862.648} C_VEL
LIN {X 0,Y 234.179,Z 744.498,A -85,B 0,C 180,E1 -19865.628,E2 -19865.628} C_VEL
LIN {X 0,Y 231.351,Z 752.825,A -85,B 0,C 180,E1 -19868.62,E2 -19868.62} C_VEL
LIN {X 0,Y 229.445,Z 758.77,A -85,B 0,C 180,E1 -19871.238,E2 -19871.238} C_VEL
LIN {X 0,Y 227.558,Z 765.315,A -85,B 0,C 180,E1 -19874.78,E2 -19874.78} C_VEL
LIN {X 0,Y 226.345,Z 770.393,A -85,B 0,C 180,E1 -19878.355,E2 -19878.355} C_VEL
LIN {X 0,Y 225.886,Z 773.336,A -85,B 0,C 180,E1 -19881.05,E2 -19881.05} C_VEL
LIN {X 0,Y 225.589,Z 776.106,A -85,B 0,C 180,E1 -19884.636,E2 -19884.636} C_VEL
LIN {X 0,Y 225.652,Z 777.671,A -85,B 0,C 180,E1 -19888.214,E2 -19888.214} C_VEL
LIN {X 0,Y 225.733,Z 778.013,A -85,B 0,C 180,E1 -19889.999,E2 -19889.999} C_VEL
LIN {X 0,Y 225.549,Z 777.821,A -85,B 0,C 180,E1 -19893.572,E2 -19893.572} C_VEL
LIN {X 0,Y 225.676,Z 776.457,A -85,B 0,C 180,E1 -19897.155,E2 -19897.155} C_VEL
LIN {X 0,Y 226.163,Z 773.896,A -85,B 0,C 180,E1 -19900.745,E2 -19900.745} C_VEL
LIN {X 0,Y 227.312,Z 770.141,A -85,B 0,C 180,E1 -19904.319,E2 -19904.319} C_VEL
LIN {X 0,Y 229.109,Z 764.851,A -85,B 0,C 180,E1 -19908.023,E2 -19908.023} C_VEL
LIN {X 0,Y 231.625,Z 758.656,A -85,B 0,C 180,E1 -19911.351,E2 -19911.351} C_VEL
LIN {X 0,Y 235.008,Z 750.634,A -85,B 0,C 180,E1 -19914.75,E2 -19914.75} C_VEL
LIN {X 0,Y 238.615,Z 742.136,A -85,B 0,C 180,E1 -19917.637,E2 -19917.637} C_VEL
LIN {X 0,Y 242.701,Z 731.947,A -85,B 0,C 180,E1 -19920.446,E2 -19920.446} C_VEL
LIN {X 0,Y 246.789,Z 721.57,A -85,B 0,C 180,E1 -19922.755,E2 -19922.755} C_VEL
LIN {X 0,Y 251.229,Z 709.18,A -85,B 0,C 180,E1 -19924.991,E2 -19924.991} C_VEL
LIN {X 0,Y 255.293,Z 696.804,A -85,B 0,C 180,E1 -19926.779,E2 -19926.779} C_VEL
LIN {X 0,Y 259.07,Z 683.343,A -85,B 0,C 180,E1 -19928.355,E2 -19928.355} C_VEL
LIN {X 0,Y 262.66,Z 668.407,A -85,B 0,C 180,E1 -19929.702,E2 -19929.702} C_VEL
LIN {X 0,Y 265.305,Z 655.339,A -85,B 0,C 180,E1 -19930.59,E2 -19930.59} C_VEL
LIN {X 0,Y 267.614,Z 640.245,A -85,B 0,C 180,E1 -19931.347,E2 -19931.347} C_VEL
LIN {X 0,Y 269.066,Z 624.672,A -85,B 0,C 180,E1 -19931.887,E2 -19931.887} C_VEL
LIN {X 0,Y 274.329,Z 540.453,A -85,B 0,C 180,E1 -19934.064,E2 -19934.064} C_VEL
LIN {X 0,Y 274.243,Z 538.891,A -85,B 0,C 180,E1 -19934.148,E2 -19934.148} C_VEL
LIN {X 0,Y 269.339,Z 527.123,A -85,B 0,C 180,E1 -19935.846,E2 -19935.846} C_VEL
LIN {X 0,Y 263.797,Z 515.619,A -85,B 0,C 180,E1 -19937.854,E2 -19937.854} C_VEL
LIN {X 0,Y 258.593,Z 506.174,A -85,B 0,C 180,E1 -19939.886,E2 -19939.886} C_VEL
LIN {X 0,Y 253.505,Z 497.661,A -85,B 0,C 180,E1 -19942.048,E2 -19942.048} C_VEL
LIN {X 0,Y 250.26,Z 492.545,A -85,B 0,C 180,E1 -19943.55,E2 -19943.55} C_VEL
LIN {X 0,Y 246.825,Z 487.243,A -85,B 0,C 180,E1 -19945.287,E2 -19945.287} C_VEL
LIN {X 0,Y 242.662,Z 481.485,A -85,B 0,C 180,E1 -19947.567,E2 -19947.567} C_VEL
LIN {X 0,Y 237.874,Z 475.023,A -85,B 0,C 180,E1 -19950.665,E2 -19950.665} C_VEL
LIN {X 0,Y 236.229,Z 473.351,A -85,B 0,C 180,E1 -19951.817,E2 -19951.817} C_VEL
LIN {X 0,Y 234.168,Z 471.004,A -85,B 0,C 180,E1 -19953.443,E2 -19953.443} C_VEL
LIN {X 0,Y 233.225,Z 468.702,A -85,B 0,C 180,E1 -19954.401,E2 -19954.401} C_VEL
LIN {X 0,Y 230.315,Z 467.212,A -85,B 0,C 180,E1 -19957.075,E2 -19957.075} C_VEL
LIN {X 0,Y 228.301,Z 464.25,A -85,B 0,C 180,E1 -19959.738,E2 -19959.738} C_VEL
LIN {X 0,Y 227.959,Z 462.707,A -85,B 0,C 180,E1 -19960.528,E2 -19960.528} C_VEL
LIN {X 0,Y 228.052,Z 462.694,A -85,B 0,C 180,E1 -19963.898,E2 -19963.898} C_VEL
LIN {X 0,Y 228.069,Z 462.692,A -85,B 0,C 180,E1 -19967.543,E2 -19967.543} C_VEL
LIN {X 0,Y 228.3,Z 462.663,A -85,B 0,C 180,E1 -19971.146,E2 -19971.146} C_VEL
LIN {X 0,Y 228.35,Z 462.661,A -85,B 0,C 180,E1 -19972.929,E2 -19972.929} C_VEL
LIN {X 0,Y 228.568,Z 462.656,A -85,B 0,C 180,E1 -19978.789,E2 -19978.789} C_VEL
LIN {X 0,Y 229.125,Z 464.582,A -85,B 0,C 180,E1 -19979.781,E2 -19979.781} C_VEL
LIN {X 0,Y 231.369,Z 467.581,A -85,B 0,C 180,E1 -19982.395,E2 -19982.395} C_VEL
LIN {X 0,Y 233.53,Z 468.883,A -85,B 0,C 180,E1 -19984.315,E2 -19984.315} C_VEL
LIN {X 0,Y 235.002,Z 471.74,A -85,B 0,C 180,E1 -19985.686,E2 -19985.686} C_VEL
LIN {X 0,Y 237.748,Z 474.097,A -85,B 0,C 180,E1 -19987.645,E2 -19987.645} C_VEL
LIN {X 0,Y 238.434,Z 474.741,A -85,B 0,C 180,E1 -19988.102,E2 -19988.102} C_VEL
LIN {X 0,Y 240.246,Z 477.803,A -85,B 0,C 180,E1 -19989.365,E2 -19989.365} C_VEL
LIN {X 0,Y 242.642,Z 480.19,A -85,B 0,C 180,E1 -19990.788,E2 -19990.788} C_VEL
LIN {X 0,Y 245.107,Z 483.695,A -85,B 0,C 180,E1 -19992.189,E2 -19992.189} C_VEL
LIN {X 0,Y 246.802,Z 485.456,A -85,B 0,C 180,E1 -19993.051,E2 -19993.051} C_VEL
LIN {X 0,Y 250.562,Z 490.646,A -85,B 0,C 180,E1 -19994.915,E2 -19994.915} C_VEL
LIN {X 0,Y 254.109,Z 495.492,A -85,B 0,C 180,E1 -19996.508,E2 -19996.508} C_VEL
LIN {X 0,Y 261.386,Z 506.051,A -85,B 0,C 180,E1 -19999.435,E2 -19999.435} C_VEL
LIN {X 0,Y 266.956,Z 515.278,A -85,B 0,C 180,E1 -20001.464,E2 -20001.464} C_VEL
LIN {X 0,Y 272.45,Z 526.474,A -85,B 0,C 180,E1 -20003.372,E2 -20003.372} C_VEL
LIN {X 0,Y 274.687,Z 531.463,A -85,B 0,C 180,E1 -20004.115,E2 -20004.115} C_VEL
LIN {X 0,Y 269.139,Z 620.258,A -85,B 0,C 180,E1 -20006.459,E2 -20006.459} C_VEL
LIN {X 0,Y 267.243,Z 636.44,A -85,B 0,C 180,E1 -20007.126,E2 -20007.126} C_VEL
LIN {X 0,Y 264.805,Z 651.517,A -85,B 0,C 180,E1 -20008.062,E2 -20008.062} C_VEL
LIN {X 0,Y 261.716,Z 666.222,A -85,B 0,C 180,E1 -20009.288,E2 -20009.288} C_VEL
LIN {X 0,Y 258.16,Z 680.099,A -85,B 0,C 180,E1 -20010.779,E2 -20010.779} C_VEL
LIN {X 0,Y 254.224,Z 693.096,A -85,B 0,C 180,E1 -20012.526,E2 -20012.526} C_VEL
LIN {X 0,Y 250.434,Z 704.466,A -85,B 0,C 180,E1 -20014.436,E2 -20014.436} C_VEL
LIN {X 0,Y 245.897,Z 716.435,A -85,B 0,C 180,E1 -20016.885,E2 -20016.885} C_VEL
LIN {X 0,Y 242.062,Z 726.041,A -85,B 0,C 180,E1 -20019.344,E2 -20019.344} C_VEL
LIN {X 0,Y 238.497,Z 734.356,A -85,B 0,C 180,E1 -20021.923,E2 -20021.923} C_VEL
LIN {X 0,Y 235.124,Z 741.913,A -85,B 0,C 180,E1 -20024.776,E2 -20024.776} C_VEL
LIN {X 0,Y 231.95,Z 749.126,A -85,B 0,C 180,E1 -20028.197,E2 -20028.197} C_VEL
LIN {X 0,Y 229.752,Z 754.119,A -85,B 0,C 180,E1 -20031.166,E2 -20031.166} C_VEL
LIN {X 0,Y 228.102,Z 758.021,A -85,B 0,C 180,E1 -20034.17,E2 -20034.17} C_VEL
LIN {X 0,Y 227.132,Z 760.592,A -85,B 0,C 180,E1 -20036.663,E2 -20036.663} C_VEL
LIN {X 0,Y 225.989,Z 763.369,A -85,B 0,C 180,E1 -20040.549,E2 -20040.549} C_VEL
LIN {X 0,Y 225.338,Z 764.846,A -85,B 0,C 180,E1 -20044.753,E2 -20044.753} C_VEL
LIN {X 0,Y 225.265,Z 764.618,A -85,B 0,C 180,E1 -20049.386,E2 -20049.386} C_VEL
LIN {X 0,Y 225.384,Z 763.743,A -85,B 0,C 180,E1 -20051.832,E2 -20051.832} C_VEL
LIN {X 0,Y 225.959,Z 761.339,A -85,B 0,C 180,E1 -20055.593,E2 -20055.593} C_VEL
LIN {X 0,Y 226.884,Z 757.655,A -85,B 0,C 180,E1 -20059.29,E2 -20059.29} C_VEL
LIN {X 0,Y 228.326,Z 752.63,A -85,B 0,C 180,E1 -20062.929,E2 -20062.929} C_VEL
LIN {X 0,Y 230.354,Z 746.15,A -85,B 0,C 180,E1 -20066.503,E2 -20066.503} C_VEL
LIN {X 0,Y 232.565,Z 739.775,A -85,B 0,C 180,E1 -20069.323,E2 -20069.323} C_VEL
LIN {X 0,Y 235.65,Z 730.687,A -85,B 0,C 180,E1 -20072.565,E2 -20072.565} C_VEL
LIN {X 0,Y 239.061,Z 720.498,A -85,B 0,C 180,E1 -20075.484,E2 -20075.484} C_VEL
LIN {X 0,Y 242.458,Z 710.038,A -85,B 0,C 180,E1 -20077.924,E2 -20077.924} C_VEL
LIN {X 0,Y 246.137,Z 697.606,A -85,B 0,C 180,E1 -20080.281,E2 -20080.281} C_VEL
LIN {X 0,Y 249.553,Z 685.091,A -85,B 0,C 180,E1 -20082.194,E2 -20082.194} C_VEL
LIN {X 0,Y 252.812,Z 671.405,A -85,B 0,C 180,E1 -20083.874,E2 -20083.874} C_VEL
LIN {X 0,Y 255.536,Z 657.526,A -85,B 0,C 180,E1 -20085.227,E2 -20085.227} C_VEL
LIN {X 0,Y 258.002,Z 642.051,A -85,B 0,C 180,E1 -20086.366,E2 -20086.366} C_VEL
LIN {X 0,Y 259.798,Z 627.006,A -85,B 0,C 180,E1 -20087.16,E2 -20087.16} C_VEL
LIN {X 0,Y 260.96,Z 611.265,A -85,B 0,C 180,E1 -20087.703,E2 -20087.703} C_VEL
LIN {X 0,Y 265.575,Z 526.542,A -85,B 0,C 180,E1 -20089.913,E2 -20089.913} C_VEL
LIN {X 0,Y 259.895,Z 513.709,A -85,B 0,C 180,E1 -20091.395,E2 -20091.395} C_VEL
LIN {X 0,Y 255.603,Z 505.585,A -85,B 0,C 180,E1 -20092.509,E2 -20092.509} C_VEL
LIN {X 0,Y 247.152,Z 491.641,A -85,B 0,C 180,E1 -20094.786,E2 -20094.786} C_VEL
LIN {X 0,Y 238.764,Z 478.936,A -85,B 0,C 180,E1 -20097.228,E2 -20097.228} C_VEL
LIN {X 0,Y 233.763,Z 471.904,A -85,B 0,C 180,E1 -20098.779,E2 -20098.779} C_VEL
LIN {X 0,Y 231.484,Z 468.626,A -85,B 0,C 180,E1 -20099.527,E2 -20099.527} C_VEL
LIN {X 0,Y 230.644,Z 467.459,A -85,B 0,C 180,E1 -20099.807,E2 -20099.807} C_VEL
LIN {X 0,Y 228.73,Z 465.249,A -85,B 0,C 180,E1 -20100.435,E2 -20100.435} C_VEL
LIN {X 0,Y 227.876,Z 462.722,A -85,B 0,C 180,E1 -20100.827,E2 -20100.827} C_VEL
LIN {X 0,Y 227.884,Z 462.711,A -85,B 0,C 180,E1 -20103.72,E2 -20103.72} C_VEL
LIN {X 0,Y 227.87,Z 462.704,A -85,B 0,C 180,E1 -20108.087,E2 -20108.087} C_VEL
LIN {X 0,Y 227.821,Z 462.719,A -85,B 0,C 180,E1 -20112.741,E2 -20112.741} C_VEL
LIN {X 0,Y 227.851,Z 462.716,A -85,B 0,C 180,E1 -20117.266,E2 -20117.266} C_VEL
LIN {X 0,Y 227.874,Z 462.722,A -85,B 0,C 180,E1 -20121.914,E2 -20121.914} C_VEL
LIN {X 0,Y 227.894,Z 462.722,A -85,B 0,C 180,E1 -20126.373,E2 -20126.373} C_VEL
LIN {X 0,Y 227.907,Z 462.7,A -85,B 0,C 180,E1 -20130.436,E2 -20130.436} C_VEL
LIN {X 0,Y 227.927,Z 462.715,A -85,B 0,C 180,E1 -20134.425,E2 -20134.425} C_VEL
LIN {X 0,Y 227.95,Z 462.701,A -85,B 0,C 180,E1 -20138.285,E2 -20138.285} C_VEL
LIN {X 0,Y 228.037,Z 462.682,A -85,B 0,C 180,E1 -20142.826,E2 -20142.826} C_VEL
LIN {X 0,Y 228.096,Z 462.694,A -85,B 0,C 180,E1 -20147.544,E2 -20147.544} C_VEL
LIN {X 0,Y 228.308,Z 462.649,A -85,B 0,C 180,E1 -20151.146,E2 -20151.146} C_VEL
LIN {X 0,Y 228.357,Z 462.662,A -85,B 0,C 180,E1 -20152.928,E2 -20152.928} C_VEL
LIN {X 0,Y 228.556,Z 462.621,A -85,B 0,C 180,E1 -20158.237,E2 -20158.237} C_VEL
LIN {X 0,Y 228.556,Z 462.634,A -85,B 0,C 180,E1 -20161.762,E2 -20161.762} C_VEL
LIN {X 0,Y 228.357,Z 462.657,A -85,B 0,C 180,E1 -20167.071,E2 -20167.071} C_VEL
LIN {X 0,Y 228.302,Z 462.668,A -85,B 0,C 180,E1 -20168.592,E2 -20168.592} C_VEL
LIN {X 0,Y 227.984,Z 462.715,A -85,B 0,C 180,E1 -20169.575,E2 -20169.575} C_VEL
LIN {X 0,Y 226.582,Z 462.892,A -85,B 0,C 180,E1 -20171.024,E2 -20171.024} C_VEL
LIN {X 0,Y 222.097,Z 463.438,A -85,B 0,C 180,E1 -20174.407,E2 -20174.407} C_VEL
LIN {X 0,Y 221.063,Z 463.572,A -85,B 0,C 180,E1 -20175.928,E2 -20175.928} C_VEL
LIN {X 0,Y 221.006,Z 463.571,A -85,B 0,C 180,E1 -20176.444,E2 -20176.444} C_VEL
LIN {X 0,Y 220.911,Z 463.583,A -85,B 0,C 180,E1 -20180.484,E2 -20180.484} C_VEL
LIN {X 0,Y 220.874,Z 463.598,A -85,B 0,C 180,E1 -20184.434,E2 -20184.434} C_VEL
LIN {X 0,Y 220.837,Z 463.597,A -85,B 0,C 180,E1 -20188.513,E2 -20188.513} C_VEL
LIN {X 0,Y 220.825,Z 463.601,A -85,B 0,C 180,E1 -20192.754,E2 -20192.754} C_VEL
LIN {X 0,Y 220.837,Z 463.64,A -85,B 0,C 180,E1 -20194.354,E2 -20194.354} C_VEL
LIN {X 0,Y 221.06,Z 464.728,A -85,B 0,C 180,E1 -20194.908,E2 -20194.908} C_VEL
LIN {X 0,Y 222.373,Z 467.158,A -85,B 0,C 180,E1 -20195.432,E2 -20195.432} C_VEL
LIN {X 0,Y 225.305,Z 471.087,A -85,B 0,C 180,E1 -20196.489,E2 -20196.489} C_VEL
LIN {X 0,Y 229.125,Z 477.165,A -85,B 0,C 180,E1 -20197.84,E2 -20197.84} C_VEL
LIN {X 0,Y 233.313,Z 483.952,A -85,B 0,C 180,E1 -20199.24,E2 -20199.24} C_VEL
LIN {X 0,Y 240.234,Z 495.769,A -85,B 0,C 180,E1 -20201.439,E2 -20201.439} C_VEL
LIN {X 0,Y 247.149,Z 508.987,A -85,B 0,C 180,E1 -20203.507,E2 -20203.507} C_VEL
LIN {X 0,Y 254.515,Z 524.703,A -85,B 0,C 180,E1 -20205.601,E2 -20205.601} C_VEL
LIN {X 0,Y 259.686,Z 537.134,A -85,B 0,C 180,E1 -20207.024,E2 -20207.024} C_VEL
LIN {X 0,Y 254.244,Z 632.938,A -85,B 0,C 180,E1 -20209.618,E2 -20209.618} C_VEL
LIN {X 0,Y 252.526,Z 648.685,A -85,B 0,C 180,E1 -20210.329,E2 -20210.329} C_VEL
LIN {X 0,Y 250.053,Z 663.786,A -85,B 0,C 180,E1 -20211.291,E2 -20211.291} C_VEL
LIN {X 0,Y 247.108,Z 678.4,A -85,B 0,C 180,E1 -20212.56,E2 -20212.56} C_VEL
LIN {X 0,Y 243.724,Z 692.555,A -85,B 0,C 180,E1 -20214.161,E2 -20214.161} C_VEL
LIN {X 0,Y 240.2,Z 705.314,A -85,B 0,C 180,E1 -20215.973,E2 -20215.973} C_VEL
LIN {X 0,Y 236.421,Z 717.664,A -85,B 0,C 180,E1 -20218.153,E2 -20218.153} C_VEL
LIN {X 0,Y 232.653,Z 728.926,A -85,B 0,C 180,E1 -20220.601,E2 -20220.601} C_VEL
LIN {X 0,Y 229.488,Z 738.422,A -85,B 0,C 180,E1 -20223.146,E2 -20223.146} C_VEL
LIN {X 0,Y 226.705,Z 746.482,A -85,B 0,C 180,E1 -20225.747,E2 -20225.747} C_VEL
LIN {X 0,Y 223.959,Z 754.429,A -85,B 0,C 180,E1 -20228.845,E2 -20228.845} C_VEL
LIN {X 0,Y 221.81,Z 760.833,A -85,B 0,C 180,E1 -20231.904,E2 -20231.904} C_VEL
LIN {X 0,Y 220.285,Z 766.383,A -85,B 0,C 180,E1 -20235.212,E2 -20235.212} C_VEL
LIN {X 0,Y 219.136,Z 771.143,A -85,B 0,C 180,E1 -20238.905,E2 -20238.905} C_VEL
LIN {X 0,Y 218.618,Z 774.584,A -85,B 0,C 180,E1 -20242.611,E2 -20242.611} C_VEL
LIN {X 0,Y 218.45,Z 776.781,A -85,B 0,C 180,E1 -20246.31,E2 -20246.31} C_VEL
LIN {X 0,Y 218.647,Z 777.796,A -85,B 0,C 180,E1 -20249.999,E2 -20249.999} C_VEL
LIN {X 0,Y 218.448,Z 777.64,A -85,B 0,C 180,E1 -20253.688,E2 -20253.688} C_VEL
LIN {X 0,Y 218.601,Z 776.294,A -85,B 0,C 180,E1 -20257.388,E2 -20257.388} C_VEL
LIN {X 0,Y 219.146,Z 773.769,A -85,B 0,C 180,E1 -20261.093,E2 -20261.093} C_VEL
LIN {X 0,Y 220.383,Z 770.053,A -85,B 0,C 180,E1 -20264.779,E2 -20264.779} C_VEL
LIN {X 0,Y 222.205,Z 765.06,A -85,B 0,C 180,E1 -20268.437,E2 -20268.437} C_VEL
LIN {X 0,Y 224.992,Z 758.674,A -85,B 0,C 180,E1 -20272.013,E2 -20272.013} C_VEL
LIN {X 0,Y 228.562,Z 750.713,A -85,B 0,C 180,E1 -20275.497,E2 -20275.497} C_VEL
LIN {X 0,Y 232.446,Z 741.889,A -85,B 0,C 180,E1 -20278.577,E2 -20278.577} C_VEL
LIN {X 0,Y 236.595,Z 732.156,A -85,B 0,C 180,E1 -20281.319,E2 -20281.319} C_VEL
LIN {X 0,Y 240.837,Z 721.869,A -85,B 0,C 180,E1 -20283.671,E2 -20283.671} C_VEL
LIN {X 0,Y 245.458,Z 709.615,A -85,B 0,C 180,E1 -20285.94,E2 -20285.94} C_VEL
LIN {X 0,Y 249.667,Z 697.384,A -85,B 0,C 180,E1 -20287.751,E2 -20287.751} C_VEL
LIN {X 0,Y 253.541,Z 684.243,A -85,B 0,C 180,E1 -20289.325,E2 -20289.325} C_VEL
LIN {X 0,Y 257.274,Z 669.458,A -85,B 0,C 180,E1 -20290.706,E2 -20290.706} C_VEL
LIN {X 0,Y 259.984,Z 656.628,A -85,B 0,C 180,E1 -20291.603,E2 -20291.603} C_VEL
LIN {X 0,Y 262.376,Z 642.13,A -85,B 0,C 180,E1 -20292.362,E2 -20292.362} C_VEL
LIN {X 0,Y 264.058,Z 626.387,A -85,B 0,C 180,E1 -20292.935,E2 -20292.935} C_VEL
LIN {X 0,Y 269.511,Z 542.713,A -85,B 0,C 180,E1 -20295.132,E2 -20295.132} C_VEL
LIN {X 0,Y 269.399,Z 541.268,A -85,B 0,C 180,E1 -20295.222,E2 -20295.222} C_VEL
LIN {X 0,Y 264.802,Z 530.259,A -85,B 0,C 180,E1 -20296.908,E2 -20296.908} C_VEL
LIN {X 0,Y 260.161,Z 520.429,A -85,B 0,C 180,E1 -20298.697,E2 -20298.697} C_VEL
LIN {X 0,Y 255.606,Z 511.867,A -85,B 0,C 180,E1 -20300.565,E2 -20300.565} C_VEL
LIN {X 0,Y 250.63,Z 503.288,A -85,B 0,C 180,E1 -20302.786,E2 -20302.786} C_VEL
LIN {X 0,Y 247.042,Z 497.512,A -85,B 0,C 180,E1 -20304.549,E2 -20304.549} C_VEL
LIN {X 0,Y 244.318,Z 493.199,A -85,B 0,C 180,E1 -20305.998,E2 -20305.998} C_VEL
LIN {X 0,Y 240.53,Z 487.727,A -85,B 0,C 180,E1 -20308.19,E2 -20308.19} C_VEL
LIN {X 0,Y 235.741,Z 481.09,A -85,B 0,C 180,E1 -20311.44,E2 -20311.44} C_VEL
LIN {X 0,Y 232.778,Z 477.965,A -85,B 0,C 180,E1 -20313.761,E2 -20313.761} C_VEL
LIN {X 0,Y 231.683,Z 475.642,A -85,B 0,C 180,E1 -20314.87,E2 -20314.87} C_VEL
LIN {X 0,Y 228.65,Z 473.681,A -85,B 0,C 180,E1 -20317.852,E2 -20317.852} C_VEL
LIN {X 0,Y 226.924,Z 470.62,A -85,B 0,C 180,E1 -20320.436,E2 -20320.436} C_VEL
LIN {X 0,Y 226.653,Z 469.689,A -85,B 0,C 180,E1 -20321,E2 -20321} C_VEL
LIN {X 0,Y 224.012,Z 468.467,A -85,B 0,C 180,E1 -20329.15,E2 -20329.15} C_VEL
LIN {X 0,Y 224.797,Z 468.873,A -85,B 0,C 180,E1 -20333.718,E2 -20333.718} C_VEL
LIN {X 0,Y 227.305,Z 469.817,A -85,B 0,C 180,E1 -20338.395,E2 -20338.395} C_VEL
LIN {X 0,Y 228.615,Z 472.767,A -85,B 0,C 180,E1 -20340.441,E2 -20340.441} C_VEL
LIN {X 0,Y 231.095,Z 475.161,A -85,B 0,C 180,E1 -20343.051,E2 -20343.051} C_VEL
LIN {X 0,Y 232.044,Z 475.885,A -85,B 0,C 180,E1 -20343.908,E2 -20343.908} C_VEL
LIN {X 0,Y 233.755,Z 478.801,A -85,B 0,C 180,E1 -20345.5,E2 -20345.5} C_VEL
LIN {X 0,Y 236.545,Z 481.324,A -85,B 0,C 180,E1 -20347.536,E2 -20347.536} C_VEL
LIN {X 0,Y 238.655,Z 484.619,A -85,B 0,C 180,E1 -20349.028,E2 -20349.028} C_VEL
LIN {X 0,Y 240.638,Z 486.724,A -85,B 0,C 180,E1 -20350.25,E2 -20350.25} C_VEL
LIN {X 0,Y 243.252,Z 490.347,A -85,B 0,C 180,E1 -20351.787,E2 -20351.787} C_VEL
LIN {X 0,Y 244.627,Z 491.911,A -85,B 0,C 180,E1 -20352.516,E2 -20352.516} C_VEL
LIN {X 0,Y 248.287,Z 497.034,A -85,B 0,C 180,E1 -20354.393,E2 -20354.393} C_VEL
LIN {X 0,Y 253.153,Z 503.87,A -85,B 0,C 180,E1 -20356.626,E2 -20356.626} C_VEL
LIN {X 0,Y 260.303,Z 514.873,A -85,B 0,C 180,E1 -20359.535,E2 -20359.535} C_VEL
LIN {X 0,Y 264.213,Z 521.937,A -85,B 0,C 180,E1 -20361.013,E2 -20361.013} C_VEL
LIN {X 0,Y 269.398,Z 533.043,A -85,B 0,C 180,E1 -20362.885,E2 -20362.885} C_VEL
LIN {X 0,Y 269.966,Z 534.402,A -85,B 0,C 180,E1 -20363.087,E2 -20363.087} C_VEL
LIN {X 0,Y 264.242,Z 620.409,A -85,B 0,C 180,E1 -20365.355,E2 -20365.355} C_VEL
LIN {X 0,Y 262.328,Z 636.281,A -85,B 0,C 180,E1 -20366.009,E2 -20366.009} C_VEL
LIN {X 0,Y 259.987,Z 650.338,A -85,B 0,C 180,E1 -20366.87,E2 -20366.87} C_VEL
LIN {X 0,Y 256.937,Z 664.79,A -85,B 0,C 180,E1 -20368.055,E2 -20368.055} C_VEL
LIN {X 0,Y 253.358,Z 678.564,A -85,B 0,C 180,E1 -20369.507,E2 -20369.507} C_VEL
LIN {X 0,Y 249.471,Z 691.153,A -85,B 0,C 180,E1 -20371.164,E2 -20371.164} C_VEL
LIN {X 0,Y 245.434,Z 702.887,A -85,B 0,C 180,E1 -20373.09,E2 -20373.09} C_VEL
LIN {X 0,Y 241.142,Z 713.974,A -85,B 0,C 180,E1 -20375.311,E2 -20375.311} C_VEL
LIN {X 0,Y 236.536,Z 725.005,A -85,B 0,C 180,E1 -20378.059,E2 -20378.059} C_VEL
LIN {X 0,Y 232.464,Z 734.18,A -85,B 0,C 180,E1 -20380.906,E2 -20380.906} C_VEL
LIN {X 0,Y 228.878,Z 741.806,A -85,B 0,C 180,E1 -20383.816,E2 -20383.816} C_VEL
LIN {X 0,Y 225.942,Z 748.178,A -85,B 0,C 180,E1 -20386.82,E2 -20386.82} C_VEL
LIN {X 0,Y 223.49,Z 753.323,A -85,B 0,C 180,E1 -20389.862,E2 -20389.862} C_VEL
LIN {X 0,Y 221.59,Z 757.466,A -85,B 0,C 180,E1 -20392.945,E2 -20392.945} C_VEL
LIN {X 0,Y 219.855,Z 761.519,A -85,B 0,C 180,E1 -20397.084,E2 -20397.084} C_VEL
LIN {X 0,Y 218.738,Z 764.029,A -85,B 0,C 180,E1 -20401.189,E2 -20401.189} C_VEL
LIN {X 0,Y 218.191,Z 765.113,A -85,B 0,C 180,E1 -20405.247,E2 -20405.247} C_VEL
LIN {X 0,Y 218.152,Z 764.847,A -85,B 0,C 180,E1 -20409.246,E2 -20409.246} C_VEL
LIN {X 0,Y 218.427,Z 763.296,A -85,B 0,C 180,E1 -20413.169,E2 -20413.169} C_VEL
LIN {X 0,Y 219.148,Z 760.47,A -85,B 0,C 180,E1 -20417.028,E2 -20417.028} C_VEL
LIN {X 0,Y 220.307,Z 756.345,A -85,B 0,C 180,E1 -20420.823,E2 -20420.823} C_VEL
LIN {X 0,Y 222.006,Z 750.844,A -85,B 0,C 180,E1 -20424.551,E2 -20424.551} C_VEL
LIN {X 0,Y 224.424,Z 743.819,A -85,B 0,C 180,E1 -20428.206,E2 -20428.206} C_VEL
LIN {X 0,Y 227.11,Z 736.252,A -85,B 0,C 180,E1 -20431.331,E2 -20431.331} C_VEL
LIN {X 0,Y 230.371,Z 727.145,A -85,B 0,C 180,E1 -20434.375,E2 -20434.375} C_VEL
LIN {X 0,Y 233.661,Z 717.571,A -85,B 0,C 180,E1 -20436.987,E2 -20436.987} C_VEL
LIN {X 0,Y 237.132,Z 706.901,A -85,B 0,C 180,E1 -20439.382,E2 -20439.382} C_VEL
LIN {X 0,Y 240.82,Z 694.889,A -85,B 0,C 180,E1 -20441.575,E2 -20441.575} C_VEL
LIN {X 0,Y 244.384,Z 681.774,A -85,B 0,C 180,E1 -20443.513,E2 -20443.513} C_VEL
LIN {X 0,Y 247.573,Z 668.141,A -85,B 0,C 180,E1 -20445.123,E2 -20445.123} C_VEL
LIN {X 0,Y 250.261,Z 654.253,A -85,B 0,C 180,E1 -20446.415,E2 -20446.415} C_VEL
LIN {X 0,Y 252.644,Z 638.704,A -85,B 0,C 180,E1 -20447.505,E2 -20447.505} C_VEL
LIN {X 0,Y 254.447,Z 623.008,A -85,B 0,C 180,E1 -20448.26,E2 -20448.26} C_VEL
LIN {X 0,Y 255.815,Z 602.163,A -85,B 0,C 180,E1 -20448.885,E2 -20448.885} C_VEL
LIN {X 0,Y 259.883,Z 528.29,A -85,B 0,C 180,E1 -20450.86,E2 -20450.86} C_VEL
LIN {X 0,Y 252.951,Z 513.345,A -85,B 0,C 180,E1 -20452.729,E2 -20452.729} C_VEL
LIN {X 0,Y 244.623,Z 499.114,A -85,B 0,C 180,E1 -20455.03,E2 -20455.03} C_VEL
LIN {X 0,Y 235.541,Z 485.042,A -85,B 0,C 180,E1 -20457.739,E2 -20457.739} C_VEL
LIN {X 0,Y 229.626,Z 476.768,A -85,B 0,C 180,E1 -20459.641,E2 -20459.641} C_VEL
LIN {X 0,Y 227.116,Z 473.117,A -85,B 0,C 180,E1 -20460.5,E2 -20460.5} C_VEL
LIN {X 0,Y 224.728,Z 469.969,A -85,B 0,C 180,E1 -20461.329,E2 -20461.329} C_VEL
LIN {X 0,Y 223.91,Z 468.582,A -85,B 0,C 180,E1 -20461.634,E2 -20461.634} C_VEL
LIN {X 0,Y 221.759,Z 466.368,A -85,B 0,C 180,E1 -20462.381,E2 -20462.381} C_VEL
LIN {X 0,Y 220.817,Z 463.586,A -85,B 0,C 180,E1 -20462.843,E2 -20462.843} C_VEL
LIN {X 0,Y 220.842,Z 463.581,A -85,B 0,C 180,E1 -20467.288,E2 -20467.288} C_VEL
LIN {X 0,Y 220.782,Z 463.601,A -85,B 0,C 180,E1 -20471.951,E2 -20471.951} C_VEL
LIN {X 0,Y 220.784,Z 463.609,A -85,B 0,C 180,E1 -20475.548,E2 -20475.548} C_VEL
LIN {X 0,Y 220.808,Z 463.595,A -85,B 0,C 180,E1 -20479.809,E2 -20479.809} C_VEL
LIN {X 0,Y 220.837,Z 463.589,A -85,B 0,C 180,E1 -20482.795,E2 -20482.795} C_VEL
LIN {X 0,Y 220.826,Z 463.604,A -85,B 0,C 180,E1 -20487.245,E2 -20487.245} C_VEL
LIN {X 0,Y 220.83,Z 463.588,A -85,B 0,C 180,E1 -20491.485,E2 -20491.485} C_VEL
LIN {X 0,Y 220.865,Z 463.578,A -85,B 0,C 180,E1 -20495.564,E2 -20495.564} C_VEL
LIN {X 0,Y 220.888,Z 463.593,A -85,B 0,C 180,E1 -20499.513,E2 -20499.513} C_VEL
LIN {X 0,Y 221.019,Z 463.554,A -85,B 0,C 180,E1 -20503.37,E2 -20503.37} C_VEL
LIN {X 0,Y 221.115,Z 463.548,A -85,B 0,C 180,E1 -20509.006,E2 -20509.006} C_VEL
LIN {X 0,Y 221.308,Z 463.538,A -85,B 0,C 180,E1 -20512.702,E2 -20512.702} C_VEL
LIN {X 0,Y 221.514,Z 463.497,A -85,B 0,C 180,E1 -20518.181,E2 -20518.181} C_VEL
LIN {X 0,Y 221.514,Z 463.51,A -85,B 0,C 180,E1 -20521.818,E2 -20521.818} C_VEL
LIN {X 0,Y 221.308,Z 463.537,A -85,B 0,C 180,E1 -20527.297,E2 -20527.297} C_VEL
LIN {X 0,Y 221.109,Z 463.543,A -85,B 0,C 180,E1 -20530.994,E2 -20530.994} C_VEL
LIN {X 0,Y 221.006,Z 463.571,A -85,B 0,C 180,E1 -20536.444,E2 -20536.444} C_VEL
LIN {X 0,Y 220.39,Z 463.651,A -85,B 0,C 180,E1 -20537.964,E2 -20537.964} C_VEL
LIN {X 0,Y 218.794,Z 463.85,A -85,B 0,C 180,E1 -20539.456,E2 -20539.456} C_VEL
LIN {X 0,Y 214.963,Z 464.33,A -85,B 0,C 180,E1 -20542.465,E2 -20542.465} C_VEL
LIN {X 0,Y 213.879,Z 464.468,A -85,B 0,C 180,E1 -20544.04,E2 -20544.04} C_VEL
LIN {X 0,Y 213.792,Z 464.472,A -85,B 0,C 180,E1 -20544.575,E2 -20544.575} C_VEL
LIN {X 0,Y 213.831,Z 464.474,A -85,B 0,C 180,E1 -20547.449,E2 -20547.449} C_VEL
LIN {X 0,Y 213.8,Z 464.486,A -85,B 0,C 180,E1 -20552.566,E2 -20552.566} C_VEL
LIN {X 0,Y 214.74,Z 467.275,A -85,B 0,C 180,E1 -20553.033,E2 -20553.033} C_VEL
LIN {X 0,Y 216.95,Z 469.557,A -85,B 0,C 180,E1 -20553.872,E2 -20553.872} C_VEL
LIN {X 0,Y 217.926,Z 471.096,A -85,B 0,C 180,E1 -20554.263,E2 -20554.263} C_VEL
LIN {X 0,Y 221.924,Z 476.87,A -85,B 0,C 180,E1 -20555.794,E2 -20555.794} C_VEL
LIN {X 0,Y 228.143,Z 486.756,A -85,B 0,C 180,E1 -20558.032,E2 -20558.032} C_VEL
LIN {X 0,Y 236.54,Z 501.408,A -85,B 0,C 180,E1 -20560.817,E2 -20560.817} C_VEL
LIN {X 0,Y 243.49,Z 515.038,A -85,B 0,C 180,E1 -20562.974,E2 -20562.974} C_VEL
LIN {X 0,Y 250.034,Z 529.378,A -85,B 0,C 180,E1 -20564.91,E2 -20564.91} C_VEL
LIN {X 0,Y 254.075,Z 539.101,A -85,B 0,C 180,E1 -20566.065,E2 -20566.065} C_VEL
LIN {X 0,Y 248.587,Z 632.614,A -85,B 0,C 180,E1 -20568.634,E2 -20568.634} C_VEL
LIN {X 0,Y 246.819,Z 648.406,A -85,B 0,C 180,E1 -20569.356,E2 -20569.356} C_VEL
LIN {X 0,Y 244.281,Z 663.532,A -85,B 0,C 180,E1 -20570.331,E2 -20570.331} C_VEL
LIN {X 0,Y 241.471,Z 677.267,A -85,B 0,C 180,E1 -20571.528,E2 -20571.528} C_VEL
LIN {X 0,Y 238.102,Z 691.029,A -85,B 0,C 180,E1 -20573.074,E2 -20573.074} C_VEL
LIN {X 0,Y 234.281,Z 704.501,A -85,B 0,C 180,E1 -20574.99,E2 -20574.99} C_VEL
LIN {X 0,Y 230.384,Z 716.963,A -85,B 0,C 180,E1 -20577.215,E2 -20577.215} C_VEL
LIN {X 0,Y 226.418,Z 728.297,A -85,B 0,C 180,E1 -20579.708,E2 -20579.708} C_VEL
LIN {X 0,Y 222.576,Z 739.308,A -85,B 0,C 180,E1 -20582.751,E2 -20582.751} C_VEL
LIN {X 0,Y 219.697,Z 747.216,A -85,B 0,C 180,E1 -20585.425,E2 -20585.425} C_VEL
LIN {X 0,Y 216.92,Z 754.996,A -85,B 0,C 180,E1 -20588.623,E2 -20588.623} C_VEL
LIN {X 0,Y 214.625,Z 761.514,A -85,B 0,C 180,E1 -20591.932,E2 -20591.932} C_VEL
LIN {X 0,Y 212.969,Z 767.309,A -85,B 0,C 180,E1 -20595.669,E2 -20595.669} C_VEL
LIN {X 0,Y 212.111,Z 770.803,A -85,B 0,C 180,E1 -20598.532,E2 -20598.532} C_VEL
LIN {X 0,Y 211.559,Z 774.288,A -85,B 0,C 180,E1 -20602.363,E2 -20602.363} C_VEL
LIN {X 0,Y 211.353,Z 776.524,A -85,B 0,C 180,E1 -20606.186,E2 -20606.186} C_VEL
LIN {X 0,Y 211.562,Z 777.579,A -85,B 0,C 180,E1 -20609.999,E2 -20609.999} C_VEL
LIN {X 0,Y 211.355,Z 777.408,A -85,B 0,C 180,E1 -20614.005,E2 -20614.005} C_VEL
LIN {X 0,Y 211.525,Z 776.13,A -85,B 0,C 180,E1 -20617.636,E2 -20617.636} C_VEL
LIN {X 0,Y 212.125,Z 773.646,A -85,B 0,C 180,E1 -20621.465,E2 -20621.465} C_VEL
LIN {X 0,Y 213.471,Z 769.978,A -85,B 0,C 180,E1 -20625.269,E2 -20625.269} C_VEL
LIN {X 0,Y 215.439,Z 765.038,A -85,B 0,C 180,E1 -20629.038,E2 -20629.038} C_VEL
LIN {X 0,Y 218.367,Z 758.7,A -85,B 0,C 180,E1 -20632.718,E2 -20632.718} C_VEL
LIN {X 0,Y 221.592,Z 751.906,A -85,B 0,C 180,E1 -20635.854,E2 -20635.854} C_VEL
LIN {X 0,Y 225.458,Z 743.784,A -85,B 0,C 180,E1 -20638.861,E2 -20638.861} C_VEL
LIN {X 0,Y 229.865,Z 733.942,A -85,B 0,C 180,E1 -20641.829,E2 -20641.829} C_VEL
LIN {X 0,Y 234.197,Z 723.98,A -85,B 0,C 180,E1 -20644.239,E2 -20644.239} C_VEL
LIN {X 0,Y 238.963,Z 712.192,A -85,B 0,C 180,E1 -20646.551,E2 -20646.551} C_VEL
LIN {X 0,Y 243.621,Z 699.399,A -85,B 0,C 180,E1 -20648.556,E2 -20648.556} C_VEL
LIN {X 0,Y 247.592,Z 686.672,A -85,B 0,C 180,E1 -20650.168,E2 -20650.168} C_VEL
LIN {X 0,Y 251.455,Z 672.366,A -85,B 0,C 180,E1 -20651.588,E2 -20651.588} C_VEL
LIN {X 0,Y 254.765,Z 657.964,A -85,B 0,C 180,E1 -20652.654,E2 -20652.654} C_VEL
LIN {X 0,Y 257.505,Z 642.35,A -85,B 0,C 180,E1 -20653.493,E2 -20653.493} C_VEL
LIN {X 0,Y 259.254,Z 626.942,A -85,B 0,C 180,E1 -20654.065,E2 -20654.065} C_VEL
LIN {X 0,Y 264.805,Z 545.338,A -85,B 0,C 180,E1 -20656.233,E2 -20656.233} C_VEL
LIN {X 0,Y 264.746,Z 543.819,A -85,B 0,C 180,E1 -20656.316,E2 -20656.316} C_VEL
LIN {X 0,Y 259.399,Z 531.096,A -85,B 0,C 180,E1 -20658.411,E2 -20658.411} C_VEL
LIN {X 0,Y 254.256,Z 520.493,A -85,B 0,C 180,E1 -20660.562,E2 -20660.562} C_VEL
LIN {X 0,Y 248.433,Z 509.891,A -85,B 0,C 180,E1 -20663.238,E2 -20663.238} C_VEL
LIN {X 0,Y 242.556,Z 500.026,A -85,B 0,C 180,E1 -20666.342,E2 -20666.342} C_VEL
LIN {X 0,Y 238.236,Z 493.767,A -85,B 0,C 180,E1 -20668.944,E2 -20668.944} C_VEL
LIN {X 0,Y 233.929,Z 487.54,A -85,B 0,C 180,E1 -20672.019,E2 -20672.019} C_VEL
LIN {X 0,Y 231.188,Z 484.558,A -85,B 0,C 180,E1 -20674.285,E2 -20674.285} C_VEL
LIN {X 0,Y 230.15,Z 482.457,A -85,B 0,C 180,E1 -20675.365,E2 -20675.365} C_VEL
LIN {X 0,Y 227.299,Z 480.373,A -85,B 0,C 180,E1 -20678.34,E2 -20678.34} C_VEL
LIN {X 0,Y 225.653,Z 477.314,A -85,B 0,C 180,E1 -20680.971,E2 -20680.971} C_VEL
LIN {X 0,Y 225.475,Z 476.667,A -85,B 0,C 180,E1 -20681.368,E2 -20681.368} C_VEL
LIN {X 0,Y 223.089,Z 475.511,A -85,B 0,C 180,E1 -20689.105,E2 -20689.105} C_VEL
LIN {X 0,Y 223.859,Z 475.892,A -85,B 0,C 180,E1 -20693.692,E2 -20693.692} C_VEL
LIN {X 0,Y 226.079,Z 476.777,A -85,B 0,C 180,E1 -20697.996,E2 -20697.996} C_VEL
LIN {X 0,Y 227.685,Z 480.068,A -85,B 0,C 180,E1 -20700.498,E2 -20700.498} C_VEL
LIN {X 0,Y 230.528,Z 482.713,A -85,B 0,C 180,E1 -20703.441,E2 -20703.441} C_VEL
LIN {X 0,Y 232.677,Z 486.014,A -85,B 0,C 180,E1 -20705.444,E2 -20705.444} C_VEL
LIN {X 0,Y 234.725,Z 487.878,A -85,B 0,C 180,E1 -20706.987,E2 -20706.987} C_VEL
LIN {X 0,Y 236.997,Z 491.338,A -85,B 0,C 180,E1 -20708.635,E2 -20708.635} C_VEL
LIN {X 0,Y 238.671,Z 493.223,A -85,B 0,C 180,E1 -20709.708,E2 -20709.708} C_VEL
LIN {X 0,Y 241.324,Z 496.894,A -85,B 0,C 180,E1 -20711.332,E2 -20711.332} C_VEL
LIN {X 0,Y 242.834,Z 498.873,A -85,B 0,C 180,E1 -20712.169,E2 -20712.169} C_VEL
LIN {X 0,Y 245.536,Z 502.643,A -85,B 0,C 180,E1 -20713.603,E2 -20713.603} C_VEL
LIN {X 0,Y 250.433,Z 509.796,A -85,B 0,C 180,E1 -20715.969,E2 -20715.969} C_VEL
LIN {X 0,Y 257.109,Z 520.307,A -85,B 0,C 180,E1 -20718.814,E2 -20718.814} C_VEL
LIN {X 0,Y 261.205,Z 528.02,A -85,B 0,C 180,E1 -20720.436,E2 -20720.436} C_VEL
LIN {X 0,Y 265.262,Z 537.147,A -85,B 0,C 180,E1 -20721.985,E2 -20721.985} C_VEL
LIN {X 0,Y 259.48,Z 620.757,A -85,B 0,C 180,E1 -20724.212,E2 -20724.212} C_VEL
LIN {X 0,Y 257.473,Z 636.646,A -85,B 0,C 180,E1 -20724.87,E2 -20724.87} C_VEL
LIN {X 0,Y 254.869,Z 651.66,A -85,B 0,C 180,E1 -20725.81,E2 -20725.81} C_VEL
LIN {X 0,Y 251.538,Z 666.432,A -85,B 0,C 180,E1 -20727.056,E2 -20727.056} C_VEL
LIN {X 0,Y 247.509,Z 681.003,A -85,B 0,C 180,E1 -20728.66,E2 -20728.66} C_VEL
LIN {X 0,Y 243.403,Z 693.571,A -85,B 0,C 180,E1 -20730.393,E2 -20730.393} C_VEL
LIN {X 0,Y 238.753,Z 706.187,A -85,B 0,C 180,E1 -20732.586,E2 -20732.586} C_VEL
LIN {X 0,Y 233.907,Z 717.831,A -85,B 0,C 180,E1 -20735.109,E2 -20735.109} C_VEL
LIN {X 0,Y 229.296,Z 728.214,A -85,B 0,C 180,E1 -20737.939,E2 -20737.939} C_VEL
LIN {X 0,Y 224.964,Z 737.239,A -85,B 0,C 180,E1 -20741,E2 -20741} C_VEL
LIN {X 0,Y 221.005,Z 745.192,A -85,B 0,C 180,E1 -20744.396,E2 -20744.396} C_VEL
LIN {X 0,Y 217.769,Z 751.68,A -85,B 0,C 180,E1 -20747.926,E2 -20747.926} C_VEL
LIN {X 0,Y 215.182,Z 756.911,A -85,B 0,C 180,E1 -20751.645,E2 -20751.645} C_VEL
LIN {X 0,Y 213.168,Z 761.224,A -85,B 0,C 180,E1 -20755.913,E2 -20755.913} C_VEL
LIN {X 0,Y 211.886,Z 763.967,A -85,B 0,C 180,E1 -20760.165,E2 -20760.165} C_VEL
LIN {X 0,Y 211.191,Z 765.275,A -85,B 0,C 180,E1 -20764.368,E2 -20764.368} C_VEL
LIN {X 0,Y 211.022,Z 765.218,A -85,B 0,C 180,E1 -20768.511,E2 -20768.511} C_VEL
LIN {X 0,Y 211.274,Z 763.85,A -85,B 0,C 180,E1 -20772.581,E2 -20772.581} C_VEL
LIN {X 0,Y 211.934,Z 761.208,A -85,B 0,C 180,E1 -20776.579,E2 -20776.579} C_VEL
LIN {X 0,Y 213.076,Z 757.275,A -85,B 0,C 180,E1 -20780.509,E2 -20780.509} C_VEL
LIN {X 0,Y 214.763,Z 751.994,A -85,B 0,C 180,E1 -20784.367,E2 -20784.367} C_VEL
LIN {X 0,Y 217.172,Z 745.227,A -85,B 0,C 180,E1 -20788.147,E2 -20788.147} C_VEL
LIN {X 0,Y 219.877,Z 737.916,A -85,B 0,C 180,E1 -20791.375,E2 -20791.375} C_VEL
LIN {X 0,Y 223.117,Z 729.127,A -85,B 0,C 180,E1 -20794.518,E2 -20794.518} C_VEL
LIN {X 0,Y 226.792,Z 719.104,A -85,B 0,C 180,E1 -20797.41,E2 -20797.41} C_VEL
LIN {X 0,Y 230.689,Z 707.643,A -85,B 0,C 180,E1 -20800.09,E2 -20800.09} C_VEL
LIN {X 0,Y 234.498,Z 695.728,A -85,B 0,C 180,E1 -20802.331,E2 -20802.331} C_VEL
LIN {X 0,Y 238.195,Z 682.726,A -85,B 0,C 180,E1 -20804.307,E2 -20804.307} C_VEL
LIN {X 0,Y 241.685,Z 668.317,A -85,B 0,C 180,E1 -20806.049,E2 -20806.049} C_VEL
LIN {X 0,Y 244.46,Z 654.482,A -85,B 0,C 180,E1 -20807.355,E2 -20807.355} C_VEL
LIN {X 0,Y 246.908,Z 638.948,A -85,B 0,C 180,E1 -20808.462,E2 -20808.462} C_VEL
LIN {X 0,Y 248.786,Z 623.241,A -85,B 0,C 180,E1 -20809.226,E2 -20809.226} C_VEL
LIN {X 0,Y 250.217,Z 602.069,A -85,B 0,C 180,E1 -20809.87,E2 -20809.87} C_VEL
LIN {X 0,Y 254.284,Z 530.533,A -85,B 0,C 180,E1 -20811.812,E2 -20811.812} C_VEL
LIN {X 0,Y 248.035,Z 517.007,A -85,B 0,C 180,E1 -20813.577,E2 -20813.577} C_VEL
LIN {X 0,Y 239.302,Z 502.041,A -85,B 0,C 180,E1 -20816.098,E2 -20816.098} C_VEL
LIN {X 0,Y 229.75,Z 487.286,A -85,B 0,C 180,E1 -20819.113,E2 -20819.113} C_VEL
LIN {X 0,Y 223.226,Z 478.271,A -85,B 0,C 180,E1 -20821.348,E2 -20821.348} C_VEL
LIN {X 0,Y 220.218,Z 474.112,A -85,B 0,C 180,E1 -20822.448,E2 -20822.448} C_VEL
LIN {X 0,Y 217.903,Z 471.128,A -85,B 0,C 180,E1 -20823.322,E2 -20823.322} C_VEL
LIN {X 0,Y 217.091,Z 469.618,A -85,B 0,C 180,E1 -20823.662,E2 -20823.662} C_VEL
LIN {X 0,Y 214.893,Z 467.524,A -85,B 0,C 180,E1 -20824.494,E2 -20824.494} C_VEL
LIN {X 0,Y 213.877,Z 465.034,A -85,B 0,C 180,E1 -20824.974,E2 -20824.974} C_VEL
LIN {X 0,Y 213.772,Z 464.484,A -85,B 0,C 180,E1 -20825.089,E2 -20825.089} C_VEL
LIN {X 0,Y 213.74,Z 464.464,A -85,B 0,C 180,E1 -20828.664,E2 -20828.664} C_VEL
LIN {X 0,Y 213.724,Z 464.489,A -85,B 0,C 180,E1 -20831.123,E2 -20831.123} C_VEL
LIN {X 0,Y 213.751,Z 464.483,A -85,B 0,C 180,E1 -20836.332,E2 -20836.332} C_VEL
LIN {X 0,Y 213.762,Z 464.485,A -85,B 0,C 180,E1 -20841.341,E2 -20841.341} C_VEL
LIN {X 0,Y 213.773,Z 464.476,A -85,B 0,C 180,E1 -20846.02,E2 -20846.02} C_VEL
LIN {X 0,Y 213.763,Z 464.461,A -85,B 0,C 180,E1 -20850.451,E2 -20850.451} C_VEL
LIN {X 0,Y 213.801,Z 464.469,A -85,B 0,C 180,E1 -20854.701,E2 -20854.701} C_VEL
LIN {X 0,Y 213.806,Z 464.47,A -85,B 0,C 180,E1 -20858.802,E2 -20858.802} C_VEL
LIN {X 0,Y 213.946,Z 464.436,A -85,B 0,C 180,E1 -20862.803,E2 -20862.803} C_VEL
LIN {X 0,Y 213.983,Z 464.454,A -85,B 0,C 180,E1 -20866.708,E2 -20866.708} C_VEL
LIN {X 0,Y 214.17,Z 464.406,A -85,B 0,C 180,E1 -20870.556,E2 -20870.556} C_VEL
LIN {X 0,Y 214.243,Z 464.414,A -85,B 0,C 180,E1 -20872.46,E2 -20872.46} C_VEL
LIN {X 0,Y 214.447,Z 464.376,A -85,B 0,C 180,E1 -20878.121,E2 -20878.121} C_VEL
LIN {X 0,Y 214.552,Z 464.384,A -85,B 0,C 180,E1 -20880,E2 -20880} C_VEL
LIN {X 0,Y 214.447,Z 464.39,A -85,B 0,C 180,E1 -20881.878,E2 -20881.878} C_VEL
LIN {X 0,Y 214.243,Z 464.419,A -85,B 0,C 180,E1 -20887.539,E2 -20887.539} C_VEL
LIN {X 0,Y 214.025,Z 464.422,A -85,B 0,C 180,E1 -20891.362,E2 -20891.362} C_VEL
LIN {X 0,Y 213.913,Z 464.45,A -85,B 0,C 180,E1 -20896.455,E2 -20896.455} C_VEL
LIN {X 0,Y 213.843,Z 464.472,A -85,B 0,C 180,E1 -20901.193,E2 -20901.193} C_VEL
LIN {X 0,Y 213.792,Z 464.472,A -85,B 0,C 180,E1 -20904.575,E2 -20904.575} C_VEL
LIN {X 0,Y 213.197,Z 464.551,A -85,B 0,C 180,E1 -20905.62,E2 -20905.62} C_VEL
LIN {X 0,Y 210.618,Z 464.88,A -85,B 0,C 180,E1 -20907.276,E2 -20907.276} C_VEL
LIN {X 0,Y 207.309,Z 465.29,A -85,B 0,C 180,E1 -20909.318,E2 -20909.318} C_VEL
LIN {X 0,Y 206.73,Z 465.358,A -85,B 0,C 180,E1 -20910.048,E2 -20910.048} C_VEL
LIN {X 0,Y 207.698,Z 468.156,A -85,B 0,C 180,E1 -20910.621,E2 -20910.621} C_VEL
LIN {X 0,Y 210.004,Z 470.486,A -85,B 0,C 180,E1 -20911.595,E2 -20911.595} C_VEL
LIN {X 0,Y 210.627,Z 471.237,A -85,B 0,C 180,E1 -20911.858,E2 -20911.858} C_VEL
LIN {X 0,Y 212.587,Z 474.295,A -85,B 0,C 180,E1 -20912.705,E2 -20912.705} C_VEL
LIN {X 0,Y 214.321,Z 476.243,A -85,B 0,C 180,E1 -20913.386,E2 -20913.386} C_VEL
LIN {X 0,Y 218.643,Z 482.672,A -85,B 0,C 180,E1 -20915.099,E2 -20915.099} C_VEL
LIN {X 0,Y 224.321,Z 491.862,A -85,B 0,C 180,E1 -20917.233,E2 -20917.233} C_VEL
LIN {X 0,Y 232.206,Z 505.821,A -85,B 0,C 180,E1 -20919.956,E2 -20919.956} C_VEL
LIN {X 0,Y 238.658,Z 518.613,A -85,B 0,C 180,E1 -20922.055,E2 -20922.055} C_VEL
LIN {X 0,Y 245.232,Z 533.154,A -85,B 0,C 180,E1 -20924.082,E2 -20924.082} C_VEL
LIN {X 0,Y 248.493,Z 541.212,A -85,B 0,C 180,E1 -20925.067,E2 -20925.067} C_VEL
LIN {X 0,Y 243.014,Z 632.097,A -85,B 0,C 180,E1 -20927.607,E2 -20927.607} C_VEL
LIN {X 0,Y 241.192,Z 648.002,A -85,B 0,C 180,E1 -20928.338,E2 -20928.338} C_VEL
LIN {X 0,Y 238.569,Z 663.174,A -85,B 0,C 180,E1 -20929.323,E2 -20929.323} C_VEL
LIN {X 0,Y 235.46,Z 677.844,A -85,B 0,C 180,E1 -20930.634,E2 -20930.634} C_VEL
LIN {X 0,Y 232.237,Z 690.619,A -85,B 0,C 180,E1 -20932.098,E2 -20932.098} C_VEL
LIN {X 0,Y 228.059,Z 704.821,A -85,B 0,C 180,E1 -20934.16,E2 -20934.16} C_VEL
LIN {X 0,Y 224.026,Z 717.197,A -85,B 0,C 180,E1 -20936.432,E2 -20936.432} C_VEL
LIN {X 0,Y 220.233,Z 727.595,A -85,B 0,C 180,E1 -20938.763,E2 -20938.763} C_VEL
LIN {X 0,Y 216.206,Z 738.724,A -85,B 0,C 180,E1 -20941.878,E2 -20941.878} C_VEL
LIN {X 0,Y 212.716,Z 747.927,A -85,B 0,C 180,E1 -20945.085,E2 -20945.085} C_VEL
LIN {X 0,Y 209.863,Z 755.547,A -85,B 0,C 180,E1 -20948.384,E2 -20948.384} C_VEL
LIN {X 0,Y 207.327,Z 762.645,A -85,B 0,C 180,E1 -20952.236,E2 -20952.236} C_VEL
LIN {X 0,Y 205.66,Z 768.208,A -85,B 0,C 180,E1 -20956.159,E2 -20956.159} C_VEL
LIN {X 0,Y 204.708,Z 772.387,A -85,B 0,C 180,E1 -20960.115,E2 -20960.115} C_VEL
LIN {X 0,Y 204.332,Z 775.281,A -85,B 0,C 180,E1 -20964.076,E2 -20964.076} C_VEL
LIN {X 0,Y 204.344,Z 776.961,A -85,B 0,C 180,E1 -20968.028,E2 -20968.028} C_VEL
LIN {X 0,Y 204.479,Z 777.362,A -85,B 0,C 180,E1 -20969.999,E2 -20969.999} C_VEL
LIN {X 0,Y 204.258,Z 777.267,A -85,B 0,C 180,E1 -20973.945,E2 -20973.945} C_VEL
LIN {X 0,Y 204.451,Z 775.973,A -85,B 0,C 180,E1 -20977.902,E2 -20977.902} C_VEL
LIN {X 0,Y 205.125,Z 773.533,A -85,B 0,C 180,E1 -20981.862,E2 -20981.862} C_VEL
LIN {X 0,Y 206.555,Z 769.909,A -85,B 0,C 180,E1 -20985.794,E2 -20985.794} C_VEL
LIN {X 0,Y 208.703,Z 765.015,A -85,B 0,C 180,E1 -20989.677,E2 -20989.677} C_VEL
LIN {X 0,Y 211.788,Z 758.735,A -85,B 0,C 180,E1 -20993.465,E2 -20993.465} C_VEL
LIN {X 0,Y 215.202,Z 751.99,A -85,B 0,C 180,E1 -20996.681,E2 -20996.681} C_VEL
LIN {X 0,Y 218.847,Z 744.746,A -85,B 0,C 180,E1 -20999.472,E2 -20999.472} C_VEL
LIN {X 0,Y 223.125,Z 735.653,A -85,B 0,C 180,E1 -21002.374,E2 -21002.374} C_VEL
LIN {X 0,Y 228.362,Z 724.291,A -85,B 0,C 180,E1 -21005.241,E2 -21005.241} C_VEL
LIN {X 0,Y 233.318,Z 712.609,A -85,B 0,C 180,E1 -21007.586,E2 -21007.586} C_VEL
LIN {X 0,Y 238.107,Z 700.063,A -85,B 0,C 180,E1 -21009.604,E2 -21009.604} C_VEL
LIN {X 0,Y 242.249,Z 687.468,A -85,B 0,C 180,E1 -21011.244,E2 -21011.244} C_VEL
LIN {X 0,Y 246.247,Z 673.446,A -85,B 0,C 180,E1 -21012.673,E2 -21012.673} C_VEL
LIN {X 0,Y 249.658,Z 659.435,A -85,B 0,C 180,E1 -21013.743,E2 -21013.743} C_VEL
LIN {X 0,Y 252.477,Z 644.49,A -85,B 0,C 180,E1 -21014.585,E2 -21014.585} C_VEL
LIN {X 0,Y 254.422,Z 629.095,A -85,B 0,C 180,E1 -21015.198,E2 -21015.198} C_VEL
LIN {X 0,Y 260.274,Z 546.704,A -85,B 0,C 180,E1 -21017.411,E2 -21017.411} C_VEL
LIN {X 0,Y 254.987,Z 533.972,A -85,B 0,C 180,E1 -21019.631,E2 -21019.631} C_VEL
LIN {X 0,Y 250.354,Z 524.282,A -85,B 0,C 180,E1 -21021.71,E2 -21021.71} C_VEL
LIN {X 0,Y 245.129,Z 514.696,A -85,B 0,C 180,E1 -21024.274,E2 -21024.274} C_VEL
LIN {X 0,Y 241.968,Z 509.266,A -85,B 0,C 180,E1 -21025.991,E2 -21025.991} C_VEL
LIN {X 0,Y 239.68,Z 505.389,A -85,B 0,C 180,E1 -21027.33,E2 -21027.33} C_VEL
LIN {X 0,Y 236.268,Z 500.123,A -85,B 0,C 180,E1 -21029.53,E2 -21029.53} C_VEL
LIN {X 0,Y 232.182,Z 494.061,A -85,B 0,C 180,E1 -21032.586,E2 -21032.586} C_VEL
LIN {X 0,Y 229.585,Z 491.091,A -85,B 0,C 180,E1 -21034.85,E2 -21034.85} C_VEL
LIN {X 0,Y 228.578,Z 489.196,A -85,B 0,C 180,E1 -21035.926,E2 -21035.926} C_VEL
LIN {X 0,Y 225.971,Z 487.106,A -85,B 0,C 180,E1 -21038.829,E2 -21038.829} C_VEL
LIN {X 0,Y 224.4,Z 483.954,A -85,B 0,C 180,E1 -21041.527,E2 -21041.527} C_VEL
LIN {X 0,Y 224.306,Z 483.647,A -85,B 0,C 180,E1 -21041.741,E2 -21041.741} C_VEL
LIN {X 0,Y 222.166,Z 482.553,A -85,B 0,C 180,E1 -21049.059,E2 -21049.059} C_VEL
LIN {X 0,Y 222.919,Z 482.929,A -85,B 0,C 180,E1 -21053.665,E2 -21053.665} C_VEL
LIN {X 0,Y 224.917,Z 483.775,A -85,B 0,C 180,E1 -21057.677,E2 -21057.677} C_VEL
LIN {X 0,Y 226.587,Z 487.12,A -85,B 0,C 180,E1 -21060.334,E2 -21060.334} C_VEL
LIN {X 0,Y 229.039,Z 489.455,A -85,B 0,C 180,E1 -21062.969,E2 -21062.969} C_VEL
LIN {X 0,Y 231.15,Z 492.719,A -85,B 0,C 180,E1 -21065.009,E2 -21065.009} C_VEL
LIN {X 0,Y 233.057,Z 494.678,A -85,B 0,C 180,E1 -21066.521,E2 -21066.521} C_VEL
LIN {X 0,Y 235.657,Z 498.375,A -85,B 0,C 180,E1 -21068.441,E2 -21068.441} C_VEL
LIN {X 0,Y 236.947,Z 500.096,A -85,B 0,C 180,E1 -21069.309,E2 -21069.309} C_VEL
LIN {X 0,Y 240.554,Z 505.043,A -85,B 0,C 180,E1 -21071.531,E2 -21071.531} C_VEL
LIN {X 0,Y 243.628,Z 509.544,A -85,B 0,C 180,E1 -21073.224,E2 -21073.224} C_VEL
LIN {X 0,Y 247.776,Z 515.709,A -85,B 0,C 180,E1 -21075.309,E2 -21075.309} C_VEL
LIN {X 0,Y 254.02,Z 525.879,A -85,B 0,C 180,E1 -21078.103,E2 -21078.103} C_VEL
LIN {X 0,Y 257.494,Z 532.581,A -85,B 0,C 180,E1 -21079.544,E2 -21079.544} C_VEL
LIN {X 0,Y 260.639,Z 539.655,A -85,B 0,C 180,E1 -21080.822,E2 -21080.822} C_VEL
LIN {X 0,Y 254.727,Z 622.144,A -85,B 0,C 180,E1 -21083.058,E2 -21083.058} C_VEL
LIN {X 0,Y 252.623,Z 637.816,A -85,B 0,C 180,E1 -21083.734,E2 -21083.734} C_VEL
LIN {X 0,Y 249.907,Z 652.629,A -85,B 0,C 180,E1 -21084.678,E2 -21084.678} C_VEL
LIN {X 0,Y 246.566,Z 666.842,A -85,B 0,C 180,E1 -21085.892,E2 -21085.892} C_VEL
LIN {X 0,Y 242.769,Z 680.171,A -85,B 0,C 180,E1 -21087.358,E2 -21087.358} C_VEL
LIN {X 0,Y 238.385,Z 693.164,A -85,B 0,C 180,E1 -21089.147,E2 -21089.147} C_VEL
LIN {X 0,Y 233.973,Z 704.686,A -85,B 0,C 180,E1 -21091.133,E2 -21091.133} C_VEL
LIN {X 0,Y 229.227,Z 715.837,A -85,B 0,C 180,E1 -21093.496,E2 -21093.496} C_VEL
LIN {X 0,Y 224.335,Z 726.41,A -85,B 0,C 180,E1 -21096.286,E2 -21096.286} C_VEL
LIN {X 0,Y 219.948,Z 735.279,A -85,B 0,C 180,E1 -21099.21,E2 -21099.21} C_VEL
LIN {X 0,Y 215.552,Z 743.645,A -85,B 0,C 180,E1 -21102.66,E2 -21102.66} C_VEL
LIN {X 0,Y 212.249,Z 749.918,A -85,B 0,C 180,E1 -21105.947,E2 -21105.947} C_VEL
LIN {X 0,Y 209.617,Z 754.864,A -85,B 0,C 180,E1 -21109.174,E2 -21109.174} C_VEL
LIN {X 0,Y 207.033,Z 759.848,A -85,B 0,C 180,E1 -21113.556,E2 -21113.556} C_VEL
LIN {X 0,Y 205.721,Z 762.515,A -85,B 0,C 180,E1 -21116.867,E2 -21116.867} C_VEL
LIN {X 0,Y 204.531,Z 764.758,A -85,B 0,C 180,E1 -21121.247,E2 -21121.247} C_VEL
LIN {X 0,Y 204.195,Z 765.36,A -85,B 0,C 180,E1 -21123.493,E2 -21123.493} C_VEL
LIN {X 0,Y 203.895,Z 765.494,A -85,B 0,C 180,E1 -21127.72,E2 -21127.72} C_VEL
LIN {X 0,Y 204.089,Z 764.335,A -85,B 0,C 180,E1 -21131.947,E2 -21131.947} C_VEL
LIN {X 0,Y 204.735,Z 761.901,A -85,B 0,C 180,E1 -21136.098,E2 -21136.098} C_VEL
LIN {X 0,Y 205.831,Z 758.185,A -85,B 0,C 180,E1 -21140.171,E2 -21140.171} C_VEL
LIN {X 0,Y 207.522,Z 753.125,A -85,B 0,C 180,E1 -21144.17,E2 -21144.17} C_VEL
LIN {X 0,Y 209.902,Z 746.603,A -85,B 0,C 180,E1 -21148.082,E2 -21148.082} C_VEL
LIN {X 0,Y 212.654,Z 739.549,A -85,B 0,C 180,E1 -21151.421,E2 -21151.421} C_VEL
LIN {X 0,Y 215.93,Z 731.052,A -85,B 0,C 180,E1 -21154.668,E2 -21154.668} C_VEL
LIN {X 0,Y 219.244,Z 722.39,A -85,B 0,C 180,E1 -21157.368,E2 -21157.368} C_VEL
LIN {X 0,Y 222.98,Z 712.156,A -85,B 0,C 180,E1 -21159.984,E2 -21159.984} C_VEL
LIN {X 0,Y 226.728,Z 701.069,A -85,B 0,C 180,E1 -21162.305,E2 -21162.305} C_VEL
LIN {X 0,Y 230.493,Z 689.069,A -85,B 0,C 180,E1 -21164.345,E2 -21164.345} C_VEL
LIN {X 0,Y 234.247,Z 675.223,A -85,B 0,C 180,E1 -21166.242,E2 -21166.242} C_VEL
LIN {X 0,Y 237.281,Z 662.014,A -85,B 0,C 180,E1 -21167.674,E2 -21167.674} C_VEL
LIN {X 0,Y 239.991,Z 647.457,A -85,B 0,C 180,E1 -21168.903,E2 -21168.903} C_VEL
LIN {X 0,Y 242.126,Z 632.527,A -85,B 0,C 180,E1 -21169.832,E2 -21169.832} C_VEL
LIN {X 0,Y 243.74,Z 616.825,A -85,B 0,C 180,E1 -21170.473,E2 -21170.473} C_VEL
LIN {X 0,Y 248.775,Z 532.76,A -85,B 0,C 180,E1 -21172.801,E2 -21172.801} C_VEL
LIN {X 0,Y 243.6,Z 521.571,A -85,B 0,C 180,E1 -21174.327,E2 -21174.327} C_VEL
LIN {X 0,Y 236.015,Z 508.332,A -85,B 0,C 180,E1 -21176.593,E2 -21176.593} C_VEL
LIN {X 0,Y 226.984,Z 494.074,A -85,B 0,C 180,E1 -21179.525,E2 -21179.525} C_VEL
LIN {X 0,Y 219.783,Z 483.817,A -85,B 0,C 180,E1 -21182.079,E2 -21182.079} C_VEL
LIN {X 0,Y 216.55,Z 479.417,A -85,B 0,C 180,E1 -21183.309,E2 -21183.309} C_VEL
LIN {X 0,Y 213.509,Z 475.229,A -85,B 0,C 180,E1 -21184.527,E2 -21184.527} C_VEL
LIN {X 0,Y 211.18,Z 472.363,A -85,B 0,C 180,E1 -21185.48,E2 -21185.48} C_VEL
LIN {X 0,Y 210.058,Z 470.521,A -85,B 0,C 180,E1 -21185.976,E2 -21185.976} C_VEL
LIN {X 0,Y 207.857,Z 468.456,A -85,B 0,C 180,E1 -21186.891,E2 -21186.891} C_VEL
LIN {X 0,Y 206.858,Z 466.174,A -85,B 0,C 180,E1 -21187.401,E2 -21187.401} C_VEL
LIN {X 0,Y 206.708,Z 465.339,A -85,B 0,C 180,E1 -21187.583,E2 -21187.583} C_VEL
LIN {X 0,Y 206.652,Z 465.365,A -85,B 0,C 180,E1 -21191.565,E2 -21191.565} C_VEL
LIN {X 0,Y 206.664,Z 465.368,A -85,B 0,C 180,E1 -21195.574,E2 -21195.574} C_VEL
LIN {X 0,Y 206.684,Z 465.353,A -85,B 0,C 180,E1 -21199.753,E2 -21199.753} C_VEL
LIN {X 0,Y 206.703,Z 465.355,A -85,B 0,C 180,E1 -21202.265,E2 -21202.265} C_VEL
LIN {X 0,Y 206.735,Z 465.339,A -85,B 0,C 180,E1 -21204.695,E2 -21204.695} C_VEL
LIN {X 0,Y 206.71,Z 465.341,A -85,B 0,C 180,E1 -21209.336,E2 -21209.336} C_VEL
LIN {X 0,Y 206.735,Z 465.358,A -85,B 0,C 180,E1 -21213.772,E2 -21213.772} C_VEL
LIN {X 0,Y 206.742,Z 465.338,A -85,B 0,C 180,E1 -21218.041,E2 -21218.041} C_VEL
LIN {X 0,Y 206.876,Z 465.321,A -85,B 0,C 180,E1 -21222.196,E2 -21222.196} C_VEL
LIN {X 0,Y 206.916,Z 465.333,A -85,B 0,C 180,E1 -21226.245,E2 -21226.245} C_VEL
LIN {X 0,Y 207.108,Z 465.285,A -85,B 0,C 180,E1 -21230.231,E2 -21230.231} C_VEL
LIN {X 0,Y 207.181,Z 465.29,A -85,B 0,C 180,E1 -21232.201,E2 -21232.201} C_VEL
LIN {X 0,Y 207.384,Z 465.255,A -85,B 0,C 180,E1 -21238.057,E2 -21238.057} C_VEL
LIN {X 0,Y 207.517,Z 465.26,A -85,B 0,C 180,E1 -21240,E2 -21240} C_VEL
LIN {X 0,Y 207.384,Z 465.268,A -85,B 0,C 180,E1 -21241.942,E2 -21241.942} C_VEL
LIN {X 0,Y 207.18,Z 465.3,A -85,B 0,C 180,E1 -21247.798,E2 -21247.798} C_VEL
LIN {X 0,Y 206.945,Z 465.302,A -85,B 0,C 180,E1 -21251.757,E2 -21251.757} C_VEL
LIN {X 0,Y 206.87,Z 465.341,A -85,B 0,C 180,E1 -21255.77,E2 -21255.77} C_VEL
LIN {X 0,Y 206.815,Z 465.329,A -85,B 0,C 180,E1 -21259.865,E2 -21259.865} C_VEL
LIN {X 0,Y 206.737,Z 465.354,A -85,B 0,C 180,E1 -21264.547,E2 -21264.547} C_VEL
LIN {X 0,Y 206.761,Z 465.355,A -85,B 0,C 180,E1 -21269.529,E2 -21269.529} C_VEL
LIN {X 0,Y 206.73,Z 465.358,A -85,B 0,C 180,E1 -21270.048,E2 -21270.048} C_VEL
LIN {X 0,Y 208.285,Z 466.445,A -85,B 0,C 180,E1 -21270.737,E2 -21270.737} C_VEL
LIN {X 0,Y 209.715,Z 468.705,A -85,B 0,C 180,E1 -21271.389,E2 -21271.389} C_VEL
LIN {X 0,Y 210.895,Z 471.746,A -85,B 0,C 180,E1 -21271.981,E2 -21271.981} C_VEL
LIN {X 0,Y 214.336,Z 484.851,A -85,B 0,C 180,E1 -21273.767,E2 -21273.767} C_VEL
LIN {X 0,Y 215.891,Z 489.176,A -85,B 0,C 180,E1 -21274.585,E2 -21274.585} C_VEL
LIN {X 0,Y 216.325,Z 489.935,A -85,B 0,C 180,E1 -21274.765,E2 -21274.765} C_VEL
LIN {X 0,Y 223.167,Z 501.595,A -85,B 0,C 180,E1 -21277.387,E2 -21277.387} C_VEL
LIN {X 0,Y 230.086,Z 514.43,A -85,B 0,C 180,E1 -21279.819,E2 -21279.819} C_VEL
LIN {X 0,Y 236.728,Z 528.393,A -85,B 0,C 180,E1 -21282.035,E2 -21282.035} C_VEL
LIN {X 0,Y 242.74,Z 542.658,A -85,B 0,C 180,E1 -21283.944,E2 -21283.944} C_VEL
LIN {X 0,Y 243.065,Z 544.228,A -85,B 0,C 180,E1 -21284.076,E2 -21284.076} C_VEL
LIN {X 0,Y 237.544,Z 631.568,A -85,B 0,C 180,E1 -21286.537,E2 -21286.537} C_VEL
LIN {X 0,Y 235.628,Z 647.589,A -85,B 0,C 180,E1 -21287.268,E2 -21287.268} C_VEL
LIN {X 0,Y 232.961,Z 662.823,A -85,B 0,C 180,E1 -21288.272,E2 -21288.272} C_VEL
LIN {X 0,Y 229.96,Z 676.603,A -85,B 0,C 180,E1 -21289.5,E2 -21289.5} C_VEL
LIN {X 0,Y 226.449,Z 690.188,A -85,B 0,C 180,E1 -21291.07,E2 -21291.07} C_VEL
LIN {X 0,Y 222.262,Z 703.925,A -85,B 0,C 180,E1 -21293.073,E2 -21293.073} C_VEL
LIN {X 0,Y 218.087,Z 716.423,A -85,B 0,C 180,E1 -21295.39,E2 -21295.39} C_VEL
LIN {X 0,Y 213.459,Z 728.627,A -85,B 0,C 180,E1 -21298.21,E2 -21298.21} C_VEL
LIN {X 0,Y 209.836,Z 738.232,A -85,B 0,C 180,E1 -21300.991,E2 -21300.991} C_VEL
LIN {X 0,Y 206.218,Z 747.372,A -85,B 0,C 180,E1 -21304.244,E2 -21304.244} C_VEL
LIN {X 0,Y 203.203,Z 755.055,A -85,B 0,C 180,E1 -21307.638,E2 -21307.638} C_VEL
LIN {X 0,Y 200.483,Z 762.209,A -85,B 0,C 180,E1 -21311.608,E2 -21311.608} C_VEL
LIN {X 0,Y 198.721,Z 767.827,A -85,B 0,C 180,E1 -21315.666,E2 -21315.666} C_VEL
LIN {X 0,Y 197.665,Z 772.054,A -85,B 0,C 180,E1 -21319.759,E2 -21319.759} C_VEL
LIN {X 0,Y 197.26,Z 774.997,A -85,B 0,C 180,E1 -21323.863,E2 -21323.863} C_VEL
LIN {X 0,Y 197.246,Z 776.72,A -85,B 0,C 180,E1 -21327.957,E2 -21327.957} C_VEL
LIN {X 0,Y 197.378,Z 777.143,A -85,B 0,C 180,E1 -21329.999,E2 -21329.999} C_VEL
LIN {X 0,Y 197.171,Z 777.07,A -85,B 0,C 180,E1 -21334.087,E2 -21334.087} C_VEL
LIN {X 0,Y 197.397,Z 775.816,A -85,B 0,C 180,E1 -21338.186,E2 -21338.186} C_VEL
LIN {X 0,Y 198.115,Z 773.418,A -85,B 0,C 180,E1 -21342.288,E2 -21342.288} C_VEL
LIN {X 0,Y 199.648,Z 769.842,A -85,B 0,C 180,E1 -21346.355,E2 -21346.355} C_VEL
LIN {X 0,Y 201.97,Z 765.01,A -85,B 0,C 180,E1 -21350.362,E2 -21350.362} C_VEL
LIN {X 0,Y 205.25,Z 758.794,A -85,B 0,C 180,E1 -21354.26,E2 -21354.26} C_VEL
LIN {X 0,Y 208.869,Z 752.078,A -85,B 0,C 180,E1 -21357.557,E2 -21357.557} C_VEL
LIN {X 0,Y 212.522,Z 745.141,A -85,B 0,C 180,E1 -21360.333,E2 -21360.333} C_VEL
LIN {X 0,Y 217.155,Z 735.889,A -85,B 0,C 180,E1 -21363.378,E2 -21363.378} C_VEL
LIN {X 0,Y 221.786,Z 726.419,A -85,B 0,C 180,E1 -21365.888,E2 -21365.888} C_VEL
LIN {X 0,Y 226.83,Z 715.226,A -85,B 0,C 180,E1 -21368.29,E2 -21368.29} C_VEL
LIN {X 0,Y 232.138,Z 702.269,A -85,B 0,C 180,E1 -21370.483,E2 -21370.483} C_VEL
LIN {X 0,Y 236.486,Z 689.976,A -85,B 0,C 180,E1 -21372.163,E2 -21372.163} C_VEL
LIN {X 0,Y 240.642,Z 676.393,A -85,B 0,C 180,E1 -21373.626,E2 -21373.626} C_VEL
LIN {X 0,Y 244.334,Z 662.053,A -85,B 0,C 180,E1 -21374.805,E2 -21374.805} C_VEL
LIN {X 0,Y 247.269,Z 648.037,A -85,B 0,C 180,E1 -21375.641,E2 -21375.641} C_VEL
LIN {X 0,Y 249.421,Z 633.368,A -85,B 0,C 180,E1 -21376.294,E2 -21376.294} C_VEL
LIN {X 0,Y 251.329,Z 611.081,A -85,B 0,C 180,E1 -21376.942,E2 -21376.942} C_VEL
LIN {X 0,Y 255.79,Z 549.308,A -85,B 0,C 180,E1 -21378.614,E2 -21378.614} C_VEL
LIN {X 0,Y 251.148,Z 537.93,A -85,B 0,C 180,E1 -21380.689,E2 -21380.689} C_VEL
LIN {X 0,Y 247.119,Z 529.268,A -85,B 0,C 180,E1 -21382.618,E2 -21382.618} C_VEL
LIN {X 0,Y 242.569,Z 520.558,A -85,B 0,C 180,E1 -21384.987,E2 -21384.987} C_VEL
LIN {X 0,Y 237.822,Z 512.039,A -85,B 0,C 180,E1 -21387.783,E2 -21387.783} C_VEL
LIN {X 0,Y 234.103,Z 506.214,A -85,B 0,C 180,E1 -21390.279,E2 -21390.279} C_VEL
LIN {X 0,Y 230.627,Z 500.78,A -85,B 0,C 180,E1 -21393.023,E2 -21393.023} C_VEL
LIN {X 0,Y 228.017,Z 497.639,A -85,B 0,C 180,E1 -21395.41,E2 -21395.41} C_VEL
LIN {X 0,Y 227.029,Z 495.952,A -85,B 0,C 180,E1 -21396.496,E2 -21396.496} C_VEL
LIN {X 0,Y 224.566,Z 493.7,A -85,B 0,C 180,E1 -21399.464,E2 -21399.464} C_VEL
LIN {X 0,Y 223.214,Z 490.709,A -85,B 0,C 180,E1 -21401.988,E2 -21401.988} C_VEL
LIN {X 0,Y 221.244,Z 489.596,A -85,B 0,C 180,E1 -21409.013,E2 -21409.013} C_VEL
LIN {X 0,Y 221.979,Z 489.967,A -85,B 0,C 180,E1 -21413.638,E2 -21413.638} C_VEL
LIN {X 0,Y 223.77,Z 490.792,A -85,B 0,C 180,E1 -21417.371,E2 -21417.371} C_VEL
LIN {X 0,Y 225.453,Z 494.082,A -85,B 0,C 180,E1 -21420.112,E2 -21420.112} C_VEL
LIN {X 0,Y 227.704,Z 496.457,A -85,B 0,C 180,E1 -21422.64,E2 -21422.64} C_VEL
LIN {X 0,Y 229.941,Z 499.726,A -85,B 0,C 180,E1 -21424.829,E2 -21424.829} C_VEL
LIN {X 0,Y 231.375,Z 501.327,A -85,B 0,C 180,E1 -21426.012,E2 -21426.012} C_VEL
LIN {X 0,Y 233.913,Z 504.977,A -85,B 0,C 180,E1 -21427.967,E2 -21427.967} C_VEL
LIN {X 0,Y 235.598,Z 507.482,A -85,B 0,C 180,E1 -21429.146,E2 -21429.146} C_VEL
LIN {X 0,Y 238.478,Z 511.447,A -85,B 0,C 180,E1 -21430.966,E2 -21430.966} C_VEL
LIN {X 0,Y 241.425,Z 515.888,A -85,B 0,C 180,E1 -21432.666,E2 -21432.666} C_VEL
LIN {X 0,Y 245.297,Z 521.92,A -85,B 0,C 180,E1 -21434.701,E2 -21434.701} C_VEL
LIN {X 0,Y 250.922,Z 531.309,A -85,B 0,C 180,E1 -21437.335,E2 -21437.335} C_VEL
LIN {X 0,Y 254.048,Z 537.556,A -85,B 0,C 180,E1 -21438.712,E2 -21438.712} C_VEL
LIN {X 0,Y 256.197,Z 542.747,A -85,B 0,C 180,E1 -21439.647,E2 -21439.647} C_VEL
LIN {X 0,Y 250.227,Z 622.288,A -85,B 0,C 180,E1 -21441.811,E2 -21441.811} C_VEL
LIN {X 0,Y 248.036,Z 638.017,A -85,B 0,C 180,E1 -21442.49,E2 -21442.49} C_VEL
LIN {X 0,Y 245.159,Z 653.104,A -85,B 0,C 180,E1 -21443.463,E2 -21443.463} C_VEL
LIN {X 0,Y 241.646,Z 667.436,A -85,B 0,C 180,E1 -21444.701,E2 -21444.701} C_VEL
LIN {X 0,Y 237.611,Z 681.014,A -85,B 0,C 180,E1 -21446.214,E2 -21446.214} C_VEL
LIN {X 0,Y 232.955,Z 694.194,A -85,B 0,C 180,E1 -21448.065,E2 -21448.065} C_VEL
LIN {X 0,Y 227.914,Z 706.736,A -85,B 0,C 180,E1 -21450.301,E2 -21450.301} C_VEL
LIN {X 0,Y 223.054,Z 717.464,A -85,B 0,C 180,E1 -21452.667,E2 -21452.667} C_VEL
LIN {X 0,Y 218.143,Z 727.53,A -85,B 0,C 180,E1 -21455.445,E2 -21455.445} C_VEL
LIN {X 0,Y 213.042,Z 737.24,A -85,B 0,C 180,E1 -21458.814,E2 -21458.814} C_VEL
LIN {X 0,Y 208.527,Z 745.317,A -85,B 0,C 180,E1 -21462.382,E2 -21462.382} C_VEL
LIN {X 0,Y 204.864,Z 751.83,A -85,B 0,C 180,E1 -21466.09,E2 -21466.09} C_VEL
LIN {X 0,Y 201.845,Z 757.075,A -85,B 0,C 180,E1 -21469.998,E2 -21469.998} C_VEL
LIN {X 0,Y 199.685,Z 761.045,A -85,B 0,C 180,E1 -21474.048,E2 -21474.048} C_VEL
LIN {X 0,Y 198.142,Z 763.897,A -85,B 0,C 180,E1 -21478.351,E2 -21478.351} C_VEL
LIN {X 0,Y 197.142,Z 765.536,A -85,B 0,C 180,E1 -21483.03,E2 -21483.03} C_VEL
LIN {X 0,Y 196.793,Z 765.768,A -85,B 0,C 180,E1 -21486.87,E2 -21486.87} C_VEL
LIN {X 0,Y 196.849,Z 765.451,A -85,B 0,C 180,E1 -21489.084,E2 -21489.084} C_VEL
LIN {X 0,Y 197.167,Z 763.862,A -85,B 0,C 180,E1 -21493.433,E2 -21493.433} C_VEL
LIN {X 0,Y 197.972,Z 761.003,A -85,B 0,C 180,E1 -21497.703,E2 -21497.703} C_VEL
LIN {X 0,Y 199.348,Z 756.839,A -85,B 0,C 180,E1 -21501.894,E2 -21501.894} C_VEL
LIN {X 0,Y 201.361,Z 751.298,A -85,B 0,C 180,E1 -21505.998,E2 -21505.998} C_VEL
LIN {X 0,Y 204.173,Z 744.218,A -85,B 0,C 180,E1 -21510.001,E2 -21510.001} C_VEL
LIN {X 0,Y 207.253,Z 736.619,A -85,B 0,C 180,E1 -21513.403,E2 -21513.403} C_VEL
LIN {X 0,Y 211.005,Z 727.442,A -85,B 0,C 180,E1 -21516.695,E2 -21516.695} C_VEL
LIN {X 0,Y 214.565,Z 718.102,A -85,B 0,C 180,E1 -21519.427,E2 -21519.427} C_VEL
LIN {X 0,Y 218.623,Z 707.045,A -85,B 0,C 180,E1 -21522.062,E2 -21522.062} C_VEL
LIN {X 0,Y 222.759,Z 694.921,A -85,B 0,C 180,E1 -21524.387,E2 -21524.387} C_VEL
LIN {X 0,Y 226.658,Z 681.964,A -85,B 0,C 180,E1 -21526.388,E2 -21526.388} C_VEL
LIN {X 0,Y 230.051,Z 668.78,A -85,B 0,C 180,E1 -21528.019,E2 -21528.019} C_VEL
LIN {X 0,Y 233.03,Z 654.849,A -85,B 0,C 180,E1 -21529.376,E2 -21529.376} C_VEL
LIN {X 0,Y 235.538,Z 640.058,A -85,B 0,C 180,E1 -21530.468,E2 -21530.468} C_VEL
LIN {X 0,Y 237.517,Z 624.727,A -85,B 0,C 180,E1 -21531.253,E2 -21531.253} C_VEL
LIN {X 0,Y 239.063,Z 604.451,A -85,B 0,C 180,E1 -21531.901,E2 -21531.901} C_VEL
LIN {X 0,Y 243.296,Z 535.126,A -85,B 0,C 180,E1 -21533.837,E2 -21533.837} C_VEL
LIN {X 0,Y 238.951,Z 525.639,A -85,B 0,C 180,E1 -21535.17,E2 -21535.17} C_VEL
LIN {X 0,Y 231.641,Z 512.73,A -85,B 0,C 180,E1 -21537.459,E2 -21537.459} C_VEL
LIN {X 0,Y 222.499,Z 498.099,A -85,B 0,C 180,E1 -21540.568,E2 -21540.568} C_VEL
LIN {X 0,Y 215.686,Z 488.454,A -85,B 0,C 180,E1 -21543.099,E2 -21543.099} C_VEL
LIN {X 0,Y 212.951,Z 484.677,A -85,B 0,C 180,E1 -21544.187,E2 -21544.187} C_VEL
LIN {X 0,Y 210.228,Z 480.906,A -85,B 0,C 180,E1 -21545.322,E2 -21545.322} C_VEL
LIN {X 0,Y 207.562,Z 477.306,A -85,B 0,C 180,E1 -21546.473,E2 -21546.473} C_VEL
LIN {X 0,Y 204.32,Z 473.397,A -85,B 0,C 180,E1 -21547.929,E2 -21547.929} C_VEL
LIN {X 0,Y 203.407,Z 471.6,A -85,B 0,C 180,E1 -21548.401,E2 -21548.401} C_VEL
LIN {X 0,Y 201.103,Z 469.747,A -85,B 0,C 180,E1 -21549.454,E2 -21549.454} C_VEL
LIN {X 0,Y 199.925,Z 467.559,A -85,B 0,C 180,E1 -21550.089,E2 -21550.089} C_VEL
LIN {X 0,Y 199.634,Z 466.239,A -85,B 0,C 180,E1 -21550.36,E2 -21550.36} C_VEL
LIN {X 0,Y 199.606,Z 466.245,A -85,B 0,C 180,E1 -21555.235,E2 -21555.235} C_VEL
LIN {X 0,Y 199.676,Z 466.238,A -85,B 0,C 180,E1 -21560.746,E2 -21560.746} C_VEL
LIN {X 0,Y 199.637,Z 466.232,A -85,B 0,C 180,E1 -21565.718,E2 -21565.718} C_VEL
LIN {X 0,Y 199.7,Z 466.227,A -85,B 0,C 180,E1 -21568.136,E2 -21568.136} C_VEL
LIN {X 0,Y 199.689,Z 466.235,A -85,B 0,C 180,E1 -21572.771,E2 -21572.771} C_VEL
LIN {X 0,Y 199.717,Z 466.207,A -85,B 0,C 180,E1 -21577.226,E2 -21577.226} C_VEL
LIN {X 0,Y 199.799,Z 466.207,A -85,B 0,C 180,E1 -21581.758,E2 -21581.758} C_VEL
LIN {X 0,Y 199.85,Z 466.208,A -85,B 0,C 180,E1 -21585.749,E2 -21585.749} C_VEL
LIN {X 0,Y 200.073,Z 466.161,A -85,B 0,C 180,E1 -21589.884,E2 -21589.884} C_VEL
LIN {X 0,Y 200.04,Z 466.192,A -85,B 0,C 180,E1 -21593.949,E2 -21593.949} C_VEL
LIN {X 0,Y 200.323,Z 466.133,A -85,B 0,C 180,E1 -21597.989,E2 -21597.989} C_VEL
LIN {X 0,Y 200.482,Z 466.136,A -85,B 0,C 180,E1 -21599.999,E2 -21599.999} C_VEL
LIN {X 0,Y 200.031,Z 466.157,A -85,B 0,C 180,E1 -21604.029,E2 -21604.029} C_VEL
LIN {X 0,Y 200.122,Z 466.182,A -85,B 0,C 180,E1 -21608.075,E2 -21608.075} C_VEL
LIN {X 0,Y 199.888,Z 466.18,A -85,B 0,C 180,E1 -21612.178,E2 -21612.178} C_VEL
LIN {X 0,Y 199.809,Z 466.214,A -85,B 0,C 180,E1 -21616.343,E2 -21616.343} C_VEL
LIN {X 0,Y 199.744,Z 466.219,A -85,B 0,C 180,E1 -21620.6,E2 -21620.6} C_VEL
LIN {X 0,Y 199.677,Z 466.235,A -85,B 0,C 180,E1 -21624.983,E2 -21624.983} C_VEL
LIN {X 0,Y 199.728,Z 466.437,A -85,B 0,C 180,E1 -21627.342,E2 -21627.342} C_VEL
LIN {X 0,Y 200.609,Z 468.885,A -85,B 0,C 180,E1 -21627.871,E2 -21627.871} C_VEL
LIN {X 0,Y 202.54,Z 471.075,A -85,B 0,C 180,E1 -21628.801,E2 -21628.801} C_VEL
LIN {X 0,Y 203.68,Z 471.94,A -85,B 0,C 180,E1 -21629.31,E2 -21629.31} C_VEL
LIN {X 0,Y 205.405,Z 474.921,A -85,B 0,C 180,E1 -21630.167,E2 -21630.167} C_VEL
LIN {X 0,Y 207.545,Z 477.241,A -85,B 0,C 180,E1 -21631.106,E2 -21631.106} C_VEL
LIN {X 0,Y 210.089,Z 480.766,A -85,B 0,C 180,E1 -21632.216,E2 -21632.216} C_VEL
LIN {X 0,Y 214.44,Z 486.781,A -85,B 0,C 180,E1 -21634,E2 -21634} C_VEL
LIN {X 0,Y 216.325,Z 489.935,A -85,B 0,C 180,E1 -21634.765,E2 -21634.765} C_VEL
LIN {X 0,Y 218.407,Z 494.363,A -85,B 0,C 180,E1 -21635.632,E2 -21635.632} C_VEL
LIN {X 0,Y 220.715,Z 502.99,A -85,B 0,C 180,E1 -21636.753,E2 -21636.753} C_VEL
LIN {X 0,Y 222.37,Z 510.157,A -85,B 0,C 180,E1 -21637.582,E2 -21637.582} C_VEL
LIN {X 0,Y 224.043,Z 515.196,A -85,B 0,C 180,E1 -21638.288,E2 -21638.288} C_VEL
LIN {X 0,Y 224.754,Z 516.741,A -85,B 0,C 180,E1 -21638.553,E2 -21638.553} C_VEL
LIN {X 0,Y 231.727,Z 531.433,A -85,B 0,C 180,E1 -21640.994,E2 -21640.994} C_VEL
LIN {X 0,Y 237.601,Z 545.415,A -85,B 0,C 180,E1 -21642.956,E2 -21642.956} C_VEL
LIN {X 0,Y 232.006,Z 632.051,A -85,B 0,C 180,E1 -21645.455,E2 -21645.455} C_VEL
LIN {X 0,Y 230.036,Z 647.814,A -85,B 0,C 180,E1 -21646.196,E2 -21646.196} C_VEL
LIN {X 0,Y 227.428,Z 662.377,A -85,B 0,C 180,E1 -21647.168,E2 -21647.168} C_VEL
LIN {X 0,Y 224.083,Z 677.131,A -85,B 0,C 180,E1 -21648.504,E2 -21648.504} C_VEL
LIN {X 0,Y 220.518,Z 690.475,A -85,B 0,C 180,E1 -21650.085,E2 -21650.085} C_VEL
LIN {X 0,Y 216.15,Z 704.222,A -85,B 0,C 180,E1 -21652.141,E2 -21652.141} C_VEL
LIN {X 0,Y 212.205,Z 715.592,A -85,B 0,C 180,E1 -21654.287,E2 -21654.287} C_VEL
LIN {X 0,Y 208.069,Z 726.152,A -85,B 0,C 180,E1 -21656.709,E2 -21656.709} C_VEL
LIN {X 0,Y 204.01,Z 736.288,A -85,B 0,C 180,E1 -21659.588,E2 -21659.588} C_VEL
LIN {X 0,Y 200.333,Z 745.567,A -85,B 0,C 180,E1 -21662.866,E2 -21662.866} C_VEL
LIN {X 0,Y 196.938,Z 753.532,A -85,B 0,C 180,E1 -21666.329,E2 -21666.329} C_VEL
LIN {X 0,Y 194.042,Z 760.822,A -85,B 0,C 180,E1 -21670.336,E2 -21670.336} C_VEL
LIN {X 0,Y 192.183,Z 766.18,A -85,B 0,C 180,E1 -21674.08,E2 -21674.08} C_VEL
LIN {X 0,Y 191.07,Z 769.747,A -85,B 0,C 180,E1 -21677.249,E2 -21677.249} C_VEL
LIN {X 0,Y 190.346,Z 773.373,A -85,B 0,C 180,E1 -21681.506,E2 -21681.506} C_VEL
LIN {X 0,Y 190.084,Z 775.743,A -85,B 0,C 180,E1 -21685.758,E2 -21685.758} C_VEL
LIN {X 0,Y 190.279,Z 776.923,A -85,B 0,C 180,E1 -21689.999,E2 -21689.999} C_VEL
LIN {X 0,Y 190.082,Z 776.872,A -85,B 0,C 180,E1 -21694.239,E2 -21694.239} C_VEL
LIN {X 0,Y 190.333,Z 775.662,A -85,B 0,C 180,E1 -21698.492,E2 -21698.492} C_VEL
LIN {X 0,Y 191.12,Z 773.314,A -85,B 0,C 180,E1 -21702.745,E2 -21702.745} C_VEL
LIN {X 0,Y 192.768,Z 769.792,A -85,B 0,C 180,E1 -21706.956,E2 -21706.956} C_VEL
LIN {X 0,Y 195.265,Z 765.013,A -85,B 0,C 180,E1 -21711.094,E2 -21711.094} C_VEL
LIN {X 0,Y 198.741,Z 758.848,A -85,B 0,C 180,E1 -21715.108,E2 -21715.108} C_VEL
LIN {X 0,Y 202.591,Z 752.177,A -85,B 0,C 180,E1 -21718.488,E2 -21718.488} C_VEL
LIN {X 0,Y 206.783,Z 744.455,A -85,B 0,C 180,E1 -21721.674,E2 -21721.674} C_VEL
LIN {X 0,Y 212.032,Z 734.691,A -85,B 0,C 180,E1 -21724.872,E2 -21724.872} C_VEL
LIN {X 0,Y 216.942,Z 725.025,A -85,B 0,C 180,E1 -21727.401,E2 -21727.401} C_VEL
LIN {X 0,Y 222.249,Z 713.598,A -85,B 0,C 180,E1 -21729.816,E2 -21729.816} C_VEL
LIN {X 0,Y 227.536,Z 701.003,A -85,B 0,C 180,E1 -21731.922,E2 -21731.922} C_VEL
LIN {X 0,Y 231.859,Z 689.163,A -85,B 0,C 180,E1 -21733.536,E2 -21733.536} C_VEL
LIN {X 0,Y 236.144,Z 675.682,A -85,B 0,C 180,E1 -21734.976,E2 -21734.976} C_VEL
LIN {X 0,Y 239.983,Z 661.25,A -85,B 0,C 180,E1 -21736.148,E2 -21736.148} C_VEL
LIN {X 0,Y 243.118,Z 646.338,A -85,B 0,C 180,E1 -21737.029,E2 -21737.029} C_VEL
LIN {X 0,Y 245.34,Z 630.973,A -85,B 0,C 180,E1 -21737.68,E2 -21737.68} C_VEL
LIN {X 0,Y 251.424,Z 553.344,A -85,B 0,C 180,E1 -21739.787,E2 -21739.787} C_VEL
LIN {X 0,Y 251.423,Z 551.928,A -85,B 0,C 180,E1 -21739.86,E2 -21739.86} C_VEL
LIN {X 0,Y 247.313,Z 541.559,A -85,B 0,C 180,E1 -21741.848,E2 -21741.848} C_VEL
LIN {X 0,Y 243.265,Z 532.907,A -85,B 0,C 180,E1 -21743.913,E2 -21743.913} C_VEL
LIN {X 0,Y 239.208,Z 524.939,A -85,B 0,C 180,E1 -21746.199,E2 -21746.199} C_VEL
LIN {X 0,Y 235.171,Z 517.497,A -85,B 0,C 180,E1 -21748.766,E2 -21748.766} C_VEL
LIN {X 0,Y 232.022,Z 512.348,A -85,B 0,C 180,E1 -21751.011,E2 -21751.011} C_VEL
LIN {X 0,Y 229.056,Z 507.436,A -85,B 0,C 180,E1 -21753.493,E2 -21753.493} C_VEL
LIN {X 0,Y 226.497,Z 504.247,A -85,B 0,C 180,E1 -21755.951,E2 -21755.951} C_VEL
LIN {X 0,Y 225.761,Z 502.857,A -85,B 0,C 180,E1 -21756.809,E2 -21756.809} C_VEL
LIN {X 0,Y 223.308,Z 500.456,A -85,B 0,C 180,E1 -21759.919,E2 -21759.919} C_VEL
LIN {X 0,Y 221.97,Z 497.556,A -85,B 0,C 180,E1 -21762.564,E2 -21762.564} C_VEL
LIN {X 0,Y 220.321,Z 496.64,A -85,B 0,C 180,E1 -21768.966,E2 -21768.966} C_VEL
LIN {X 0,Y 220.911,Z 496.872,A -85,B 0,C 180,E1 -21773.149,E2 -21773.149} C_VEL
LIN {X 0,Y 222.616,Z 497.727,A -85,B 0,C 180,E1 -21777.023,E2 -21777.023} C_VEL
LIN {X 0,Y 224.487,Z 501.275,A -85,B 0,C 180,E1 -21780.113,E2 -21780.113} C_VEL
LIN {X 0,Y 226.266,Z 503.19,A -85,B 0,C 180,E1 -21782.17,E2 -21782.17} C_VEL
LIN {X 0,Y 228.639,Z 506.664,A -85,B 0,C 180,E1 -21784.567,E2 -21784.567} C_VEL
LIN {X 0,Y 229.778,Z 508.066,A -85,B 0,C 180,E1 -21785.552,E2 -21785.552} C_VEL
LIN {X 0,Y 233.067,Z 512.964,A -85,B 0,C 180,E1 -21788.139,E2 -21788.139} C_VEL
LIN {X 0,Y 236.708,Z 518.238,A -85,B 0,C 180,E1 -21790.564,E2 -21790.564} C_VEL
LIN {X 0,Y 242.169,Z 526.83,A -85,B 0,C 180,E1 -21793.704,E2 -21793.704} C_VEL
LIN {X 0,Y 247.998,Z 536.94,A -85,B 0,C 180,E1 -21796.603,E2 -21796.603} C_VEL
LIN {X 0,Y 250.953,Z 543.256,A -85,B 0,C 180,E1 -21797.99,E2 -21797.99} C_VEL
LIN {X 0,Y 251.822,Z 545.155,A -85,B 0,C 180,E1 -21798.382,E2 -21798.382} C_VEL
LIN {X 0,Y 247.607,Z 601.086,A -85,B 0,C 180,E1 -21799.899,E2 -21799.899} C_VEL
LIN {X 0,Y 245.632,Z 624.416,A -85,B 0,C 180,E1 -21800.591,E2 -21800.591} C_VEL
LIN {X 0,Y 243.43,Z 639.274,A -85,B 0,C 180,E1 -21801.258,E2 -21801.258} C_VEL
LIN {X 0,Y 240.394,Z 654.343,A -85,B 0,C 180,E1 -21802.251,E2 -21802.251} C_VEL
LIN {X 0,Y 236.659,Z 668.776,A -85,B 0,C 180,E1 -21803.529,E2 -21803.529} C_VEL
LIN {X 0,Y 232.539,Z 681.959,A -85,B 0,C 180,E1 -21805.032,E2 -21805.032} C_VEL
LIN {X 0,Y 227.728,Z 694.912,A -85,B 0,C 180,E1 -21806.882,E2 -21806.882} C_VEL
LIN {X 0,Y 222.888,Z 706.485,A -85,B 0,C 180,E1 -21808.958,E2 -21808.958} C_VEL
LIN {X 0,Y 217.639,Z 717.667,A -85,B 0,C 180,E1 -21811.451,E2 -21811.451} C_VEL
LIN {X 0,Y 212.519,Z 727.643,A -85,B 0,C 180,E1 -21814.237,E2 -21814.237} C_VEL
LIN {X 0,Y 207.204,Z 737.272,A -85,B 0,C 180,E1 -21817.628,E2 -21817.628} C_VEL
LIN {X 0,Y 202.417,Z 745.374,A -85,B 0,C 180,E1 -21821.277,E2 -21821.277} C_VEL
LIN {X 0,Y 198.517,Z 751.896,A -85,B 0,C 180,E1 -21825.077,E2 -21825.077} C_VEL
LIN {X 0,Y 194.975,Z 757.697,A -85,B 0,C 180,E1 -21829.549,E2 -21829.549} C_VEL
LIN {X 0,Y 192.458,Z 761.951,A -85,B 0,C 180,E1 -21834.25,E2 -21834.25} C_VEL
LIN {X 0,Y 190.843,Z 764.651,A -85,B 0,C 180,E1 -21838.967,E2 -21838.967} C_VEL
LIN {X 0,Y 189.968,Z 765.918,A -85,B 0,C 180,E1 -21843.646,E2 -21843.646} C_VEL
LIN {X 0,Y 189.752,Z 765.826,A -85,B 0,C 180,E1 -21848.263,E2 -21848.263} C_VEL
LIN {X 0,Y 189.976,Z 764.428,A -85,B 0,C 180,E1 -21852.787,E2 -21852.787} C_VEL
LIN {X 0,Y 190.733,Z 761.746,A -85,B 0,C 180,E1 -21857.229,E2 -21857.229} C_VEL
LIN {X 0,Y 192.09,Z 757.769,A -85,B 0,C 180,E1 -21861.586,E2 -21861.586} C_VEL
LIN {X 0,Y 194.101,Z 752.439,A -85,B 0,C 180,E1 -21865.848,E2 -21865.848} C_VEL
LIN {X 0,Y 196.915,Z 745.617,A -85,B 0,C 180,E1 -21870.001,E2 -21870.001} C_VEL
LIN {X 0,Y 200.038,Z 738.242,A -85,B 0,C 180,E1 -21873.526,E2 -21873.526} C_VEL
LIN {X 0,Y 203.805,Z 729.364,A -85,B 0,C 180,E1 -21876.933,E2 -21876.933} C_VEL
LIN {X 0,Y 207.486,Z 720.339,A -85,B 0,C 180,E1 -21879.752,E2 -21879.752} C_VEL
LIN {X 0,Y 211.606,Z 709.679,A -85,B 0,C 180,E1 -21882.468,E2 -21882.468} C_VEL
LIN {X 0,Y 215.79,Z 698.043,A -85,B 0,C 180,E1 -21884.862,E2 -21884.862} C_VEL
LIN {X 0,Y 220.069,Z 684.681,A -85,B 0,C 180,E1 -21887.061,E2 -21887.061} C_VEL
LIN {X 0,Y 223.708,Z 671.524,A -85,B 0,C 180,E1 -21888.786,E2 -21888.786} C_VEL
LIN {X 0,Y 227.005,Z 657.138,A -85,B 0,C 180,E1 -21890.266,E2 -21890.266} C_VEL
LIN {X 0,Y 229.735,Z 642.251,A -85,B 0,C 180,E1 -21891.42,E2 -21891.42} C_VEL
LIN {X 0,Y 231.842,Z 626.833,A -85,B 0,C 180,E1 -21892.268,E2 -21892.268} C_VEL
LIN {X 0,Y 233.19,Z 611.015,A -85,B 0,C 180,E1 -21892.833,E2 -21892.833} C_VEL
LIN {X 0,Y 237.97,Z 537.447,A -85,B 0,C 180,E1 -21894.889,E2 -21894.889} C_VEL
LIN {X 0,Y 234.013,Z 529.048,A -85,B 0,C 180,E1 -21896.157,E2 -21896.157} C_VEL
LIN {X 0,Y 226.718,Z 516.195,A -85,B 0,C 180,E1 -21898.546,E2 -21898.546} C_VEL
LIN {X 0,Y 218.711,Z 503.182,A -85,B 0,C 180,E1 -21901.407,E2 -21901.407} C_VEL
LIN {X 0,Y 210.3,Z 491.009,A -85,B 0,C 180,E1 -21904.723,E2 -21904.723} C_VEL
LIN {X 0,Y 206.282,Z 485.703,A -85,B 0,C 180,E1 -21906.441,E2 -21906.441} C_VEL
LIN {X 0,Y 203.696,Z 482.13,A -85,B 0,C 180,E1 -21907.629,E2 -21907.629} C_VEL
LIN {X 0,Y 201.113,Z 478.792,A -85,B 0,C 180,E1 -21908.861,E2 -21908.861} C_VEL
LIN {X 0,Y 200.237,Z 477.557,A -85,B 0,C 180,E1 -21909.301,E2 -21909.301} C_VEL
LIN {X 0,Y 197.698,Z 474.84,A -85,B 0,C 180,E1 -21910.551,E2 -21910.551} C_VEL
LIN {X 0,Y 196.394,Z 472.573,A -85,B 0,C 180,E1 -21911.28,E2 -21911.28} C_VEL
LIN {X 0,Y 193.853,Z 470.453,A -85,B 0,C 180,E1 -21912.605,E2 -21912.605} C_VEL
LIN {X 0,Y 192.697,Z 468.025,A -85,B 0,C 180,E1 -21913.346,E2 -21913.346} C_VEL
LIN {X 0,Y 192.503,Z 467.115,A -85,B 0,C 180,E1 -21913.594,E2 -21913.594} C_VEL
LIN {X 0,Y 192.537,Z 467.117,A -85,B 0,C 180,E1 -21916.891,E2 -21916.891} C_VEL
LIN {X 0,Y 192.589,Z 467.119,A -85,B 0,C 180,E1 -21921.656,E2 -21921.656} C_VEL
LIN {X 0,Y 192.602,Z 467.119,A -85,B 0,C 180,E1 -21926.814,E2 -21926.814} C_VEL
LIN {X 0,Y 192.664,Z 467.096,A -85,B 0,C 180,E1 -21931.691,E2 -21931.691} C_VEL
LIN {X 0,Y 192.688,Z 467.082,A -85,B 0,C 180,E1 -21936.346,E2 -21936.346} C_VEL
LIN {X 0,Y 192.735,Z 467.09,A -85,B 0,C 180,E1 -21941.458,E2 -21941.458} C_VEL
LIN {X 0,Y 192.774,Z 467.081,A -85,B 0,C 180,E1 -21945.214,E2 -21945.214} C_VEL
LIN {X 0,Y 192.984,Z 467.045,A -85,B 0,C 180,E1 -21949.508,E2 -21949.508} C_VEL
LIN {X 0,Y 193.071,Z 467.039,A -85,B 0,C 180,E1 -21951.627,E2 -21951.627} C_VEL
LIN {X 0,Y 193.265,Z 467.012,A -85,B 0,C 180,E1 -21957.915,E2 -21957.915} C_VEL
LIN {X 0,Y 193.446,Z 467.012,A -85,B 0,C 180,E1 -21959.999,E2 -21959.999} C_VEL
LIN {X 0,Y 192.978,Z 467.035,A -85,B 0,C 180,E1 -21964.176,E2 -21964.176} C_VEL
LIN {X 0,Y 193.071,Z 467.061,A -85,B 0,C 180,E1 -21968.372,E2 -21968.372} C_VEL
LIN {X 0,Y 192.812,Z 467.062,A -85,B 0,C 180,E1 -21972.632,E2 -21972.632} C_VEL
LIN {X 0,Y 192.774,Z 467.081,A -85,B 0,C 180,E1 -21976.957,E2 -21976.957} C_VEL
LIN {X 0,Y 192.67,Z 467.111,A -85,B 0,C 180,E1 -21981.393,E2 -21981.393} C_VEL
LIN {X 0,Y 192.7,Z 467.272,A -85,B 0,C 180,E1 -21984.191,E2 -21984.191} C_VEL
LIN {X 0,Y 193.491,Z 469.647,A -85,B 0,C 180,E1 -21984.753,E2 -21984.753} C_VEL
LIN {X 0,Y 195.246,Z 471.787,A -85,B 0,C 180,E1 -21985.734,E2 -21985.734} C_VEL
LIN {X 0,Y 196.8,Z 472.894,A -85,B 0,C 180,E1 -21986.512,E2 -21986.512} C_VEL
LIN {X 0,Y 198.713,Z 476.098,A -85,B 0,C 180,E1 -21987.555,E2 -21987.555} C_VEL
LIN {X 0,Y 200.896,Z 478.309,A -85,B 0,C 180,E1 -21988.601,E2 -21988.601} C_VEL
LIN {X 0,Y 203.449,Z 481.843,A -85,B 0,C 180,E1 -21989.84,E2 -21989.84} C_VEL
LIN {X 0,Y 204.725,Z 483.444,A -85,B 0,C 180,E1 -21990.43,E2 -21990.43} C_VEL
LIN {X 0,Y 208.767,Z 489.01,A -85,B 0,C 180,E1 -21992.229,E2 -21992.229} C_VEL
LIN {X 0,Y 211.505,Z 493.134,A -85,B 0,C 180,E1 -21993.39,E2 -21993.39} C_VEL
LIN {X 0,Y 219.017,Z 505.976,A -85,B 0,C 180,E1 -21996.415,E2 -21996.415} C_VEL
LIN {X 0,Y 224.754,Z 516.741,A -85,B 0,C 180,E1 -21998.553,E2 -21998.553} C_VEL
LIN {X 0,Y 226.581,Z 521.602,A -85,B 0,C 180,E1 -21999.261,E2 -21999.261} C_VEL
LIN {X 0,Y 228.352,Z 530.712,A -85,B 0,C 180,E1 -22000.131,E2 -22000.131} C_VEL
LIN {X 0,Y 230.295,Z 541.883,A -85,B 0,C 180,E1 -22001.115,E2 -22001.115} C_VEL
LIN {X 0,Y 231.364,Z 545.348,A -85,B 0,C 180,E1 -22001.526,E2 -22001.526} C_VEL
LIN {X 0,Y 232.331,Z 547.855,A -85,B 0,C 180,E1 -22001.865,E2 -22001.865} C_VEL
LIN {X 0,Y 226.664,Z 631.456,A -85,B 0,C 180,E1 -22004.287,E2 -22004.287} C_VEL
LIN {X 0,Y 224.669,Z 647.2,A -85,B 0,C 180,E1 -22005.027,E2 -22005.027} C_VEL
LIN {X 0,Y 221.98,Z 661.852,A -85,B 0,C 180,E1 -22006.008,E2 -22006.008} C_VEL
LIN {X 0,Y 218.744,Z 675.713,A -85,B 0,C 180,E1 -22007.255,E2 -22007.255} C_VEL
LIN {X 0,Y 215.088,Z 689.122,A -85,B 0,C 180,E1 -22008.837,E2 -22008.837} C_VEL
LIN {X 0,Y 210.951,Z 701.917,A -85,B 0,C 180,E1 -22010.727,E2 -22010.727} C_VEL
LIN {X 0,Y 206.382,Z 714.693,A -85,B 0,C 180,E1 -22013.116,E2 -22013.116} C_VEL
LIN {X 0,Y 202.102,Z 725.373,A -85,B 0,C 180,E1 -22015.591,E2 -22015.591} C_VEL
LIN {X 0,Y 198.007,Z 735.225,A -85,B 0,C 180,E1 -22018.412,E2 -22018.412} C_VEL
LIN {X 0,Y 193.968,Z 744.97,A -85,B 0,C 180,E1 -22021.898,E2 -22021.898} C_VEL
LIN {X 0,Y 190.386,Z 753.011,A -85,B 0,C 180,E1 -22025.462,E2 -22025.462} C_VEL
LIN {X 0,Y 187.587,Z 759.681,A -85,B 0,C 180,E1 -22029.15,E2 -22029.15} C_VEL
LIN {X 0,Y 185.3,Z 765.786,A -85,B 0,C 180,E1 -22033.473,E2 -22033.473} C_VEL
LIN {X 0,Y 183.824,Z 770.462,A -85,B 0,C 180,E1 -22037.86,E2 -22037.86} C_VEL
LIN {X 0,Y 183.275,Z 773.058,A -85,B 0,C 180,E1 -22041.176,E2 -22041.176} C_VEL
LIN {X 0,Y 183.012,Z 775.478,A -85,B 0,C 180,E1 -22045.594,E2 -22045.594} C_VEL
LIN {X 0,Y 183.183,Z 776.697,A -85,B 0,C 180,E1 -22049.999,E2 -22049.999} C_VEL
LIN {X 0,Y 183.01,Z 776.675,A -85,B 0,C 180,E1 -22054.404,E2 -22054.404} C_VEL
LIN {X 0,Y 183.267,Z 775.513,A -85,B 0,C 180,E1 -22058.822,E2 -22058.822} C_VEL
LIN {X 0,Y 184.139,Z 773.213,A -85,B 0,C 180,E1 -22063.237,E2 -22063.237} C_VEL
LIN {X 0,Y 185.916,Z 769.742,A -85,B 0,C 180,E1 -22067.601,E2 -22067.601} C_VEL
LIN {X 0,Y 188.61,Z 765.019,A -85,B 0,C 180,E1 -22071.876,E2 -22071.876} C_VEL
LIN {X 0,Y 192.268,Z 758.912,A -85,B 0,C 180,E1 -22076.015,E2 -22076.015} C_VEL
LIN {X 0,Y 196.37,Z 752.303,A -85,B 0,C 180,E1 -22079.477,E2 -22079.477} C_VEL
LIN {X 0,Y 201.183,Z 743.9,A -85,B 0,C 180,E1 -22083.029,E2 -22083.029} C_VEL
LIN {X 0,Y 206.225,Z 734.974,A -85,B 0,C 180,E1 -22086.004,E2 -22086.004} C_VEL
LIN {X 0,Y 212.254,Z 723.655,A -85,B 0,C 180,E1 -22088.983,E2 -22088.983} C_VEL
LIN {X 0,Y 217.841,Z 712.034,A -85,B 0,C 180,E1 -22091.403,E2 -22091.403} C_VEL
LIN {X 0,Y 223.047,Z 699.906,A -85,B 0,C 180,E1 -22093.413,E2 -22093.413} C_VEL
LIN {X 0,Y 228,Z 686.681,A -85,B 0,C 180,E1 -22095.149,E2 -22095.149} C_VEL
LIN {X 0,Y 232.335,Z 673.054,A -85,B 0,C 180,E1 -22096.549,E2 -22096.549} C_VEL
LIN {X 0,Y 236.053,Z 659.171,A -85,B 0,C 180,E1 -22097.622,E2 -22097.622} C_VEL
LIN {X 0,Y 239.154,Z 644.428,A -85,B 0,C 180,E1 -22098.454,E2 -22098.454} C_VEL
LIN {X 0,Y 241.267,Z 629.514,A -85,B 0,C 180,E1 -22099.071,E2 -22099.071} C_VEL
LIN {X 0,Y 247.228,Z 556.09,A -85,B 0,C 180,E1 -22101.068,E2 -22101.068} C_VEL
LIN {X 0,Y 247.232,Z 554.608,A -85,B 0,C 180,E1 -22101.148,E2 -22101.148} C_VEL
LIN {X 0,Y 243.183,Z 544.427,A -85,B 0,C 180,E1 -22103.244,E2 -22103.244} C_VEL
LIN {X 0,Y 239.264,Z 535.78,A -85,B 0,C 180,E1 -22105.447,E2 -22105.447} C_VEL
LIN {X 0,Y 234.89,Z 527.174,A -85,B 0,C 180,E1 -22108.174,E2 -22108.174} C_VEL
LIN {X 0,Y 232.614,Z 522.955,A -85,B 0,C 180,E1 -22109.757,E2 -22109.757} C_VEL
LIN {X 0,Y 229.938,Z 518.367,A -85,B 0,C 180,E1 -22111.818,E2 -22111.818} C_VEL
LIN {X 0,Y 227.431,Z 514.025,A -85,B 0,C 180,E1 -22114.044,E2 -22114.044} C_VEL
LIN {X 0,Y 225.005,Z 510.843,A -85,B 0,C 180,E1 -22116.499,E2 -22116.499} C_VEL
LIN {X 0,Y 224.254,Z 509.602,A -85,B 0,C 180,E1 -22117.392,E2 -22117.392} C_VEL
LIN {X 0,Y 221.86,Z 506.839,A -85,B 0,C 180,E1 -22120.746,E2 -22120.746} C_VEL
LIN {X 0,Y 220.888,Z 504.55,A -85,B 0,C 180,E1 -22122.875,E2 -22122.875} C_VEL
LIN {X 0,Y 219.399,Z 503.683,A -85,B 0,C 180,E1 -22128.919,E2 -22128.919} C_VEL
LIN {X 0,Y 219.852,Z 503.828,A -85,B 0,C 180,E1 -22132.654,E2 -22132.654} C_VEL
LIN {X 0,Y 221.515,Z 504.766,A -85,B 0,C 180,E1 -22136.766,E2 -22136.766} C_VEL
LIN {X 0,Y 223.319,Z 508.198,A -85,B 0,C 180,E1 -22139.837,E2 -22139.837} C_VEL
LIN {X 0,Y 224.865,Z 509.973,A -85,B 0,C 180,E1 -22141.72,E2 -22141.72} C_VEL
LIN {X 0,Y 227.503,Z 513.747,A -85,B 0,C 180,E1 -22144.444,E2 -22144.444} C_VEL
LIN {X 0,Y 231.031,Z 519.075,A -85,B 0,C 180,E1 -22147.417,E2 -22147.417} C_VEL
LIN {X 0,Y 234.649,Z 524.574,A -85,B 0,C 180,E1 -22149.96,E2 -22149.96} C_VEL
LIN {X 0,Y 239.596,Z 532.673,A -85,B 0,C 180,E1 -22152.957,E2 -22152.957} C_VEL
LIN {X 0,Y 244.945,Z 542.27,A -85,B 0,C 180,E1 -22155.771,E2 -22155.771} C_VEL
LIN {X 0,Y 247.675,Z 548.306,A -85,B 0,C 180,E1 -22157.121,E2 -22157.121} C_VEL
